// TwinCAT 3 PLC project MotionControl
// ProgramVersion: 3.1.4026.24
// libraries:
//   Tc2_MC2, * (Beckhoff Automation GmbH)
//   Tc2_Standard, * (Beckhoff Automation GmbH)
//   Tc2_SUPS, * (Beckhoff Automation GmbH)
//   Tc2_System, * (Beckhoff Automation GmbH)
//   Tc2_Utilities, * (Beckhoff Automation GmbH)
//   Tc3_DriveMotionControl, * (Beckhoff Automation GmbH)
//   Tc3_IotBase, * (Beckhoff Automation GmbH)
//   Tc3_JsonXml, * (Beckhoff Automation GmbH)
//   Tc3_Module, * (Beckhoff Automation GmbH)
//   VisuDialogs, * (System)
// project tree:
//   / CSVTask.TcTTO, GlobalTextList.TcGTLO, PlcTask.TcTTO, Visualization Manager.TcVMO (not stored)
//   DUTs/ BASIN.TcDUT, BasinStateDisp.TcDUT, HB.TcDUT, MotionType.TcDUT, CTR_SIGNALS_INTERNAL.TcDUT, MOTION_INSTRUCTION.TcDUT, MOTION_FB_STATUS.TcDUT, OUT_SIGNALS.TcDUT, MOTION_CTR.TcDUT, SCRIPTNAME.TcDUT, STATUS.TcDUT
//   GVLs/ GVL_MOTION.TcGVL
//   POUs/ AddCommand.TcPOU, DeleteLastInstruction.TcPOU, ClearScript.TcPOU, DeleteScriptFile.TcPOU, DirectMotion.TcPOU, HomeFixRack.TcPOU, HomeX.TcPOU, HomeY.TcPOU, HomeZ.TcPOU, JsonSaxHandler.TcPOU, MAIN.TcPOU, FunctionBlockMisc.TcPOU, AxisFunctionBlocks.TcPOU, MQTTCOMM.TcPOU, RackCheck.TcPOU, ScriptList.TcPOU, ScriptRead.TcPOU, CSVWrite.TcPOU, ResetAxes.TcPOU, RunCommands.TcPOU, zAxisMoreLogic.TcPOU
//   VISUs/ visMotorControl.TcVIS
// real-time tasks:
//   TASK PlcTask: cycle T#1ms, priority 6, ADS port 350
//   TASK VISU_TASK: cycle T#50000us, priority 14, ADS port 351
//   TASK CSVTask: cycle T#1ms, priority 8, ADS port 353
// motion (NC):
//   TASK NC-Task 1 SAF: cycle T#1ms, priority 4, ADS port 501
//   TASK NC-Task 1 SVB: cycle T#10ms, priority 12, ADS port 511
//   AXIS xAxis (id 1)
//     Dynamic: Acceleration=100, Deceleration=1000, Jerk=4000
//     Velo: RefSearch=10, RefSync=9, FastManual=250, Fast=904.22, Maximum=904.22
//     OtherSettings: AllowMotionCmdToSlave=true, DataPersistence=true
//     encoder EncType=19
//       EncPara: ScaleFactorNumerator=0.0007056311621, MaxCount=#xffffffff
//         Inc: RefSearchInverse=true, RefSyncInverse=false
//     drive DrvType=16
//       DrvPara: MaxCount=#xffffffff, DriveControlDWord=#x00020100
//         Analog: VeloReferenz=994.642, TorqueSetpointScale=10, ScaleFactorActTorque=0.1
//         TimeComp: TaskDelayCycles=1
//     controller CtrType=1
//       CtrPara: PriorControlFactor=1
//         Observer: BandWidth=20
//   AXIS yAxis (id 2)
//     Dynamic: Acceleration=200, Deceleration=2000, Jerk=6000
//     Velo: RefSearch=12, RefSync=5, SlowManual=70, FastManual=300, Fast=452.11, Maximum=452.11
//     OtherSettings: AllowMotionCmdToSlave=true, DataPersistence=true
//     encoder EncType=19
//       EncPara: ScaleFactorNumerator=0.0003125, Inverse=true, MaxCount=#xffffffff
//         Inc: RefSearchInverse=true, RefSyncInverse=false
//     drive DrvType=16
//       DrvPara: Inverse=true, MaxCount=#xffffffff, DriveControlDWord=#x00020100
//         Analog: VeloReferenz=497.321, VeloScale=32, TorqueSetpointScale=10, ScaleFactorActTorque=0.1
//         TimeComp: TaskDelayCycles=1
//     controller CtrType=1
//       CtrPara: PriorControlFactor=1
//         PosDiffControl: Range=10
//         Observer: BandWidth=20
//   AXIS xAxisCoupled (id 3)
//     Dynamic: Acceleration=100, Deceleration=1000, Jerk=4000
//     Velo: RefSearch=10, RefSync=9.0422, SlowManual=45.211, FastManual=271.266, Fast=904.22, Maximum=904.22
//     OtherSettings: AllowMotionCmdToSlave=true, DataPersistence=true
//     encoder EncType=19
//       EncPara: ScaleFactorNumerator=0.0007056311621, Inverse=true, MaxCount=#xffffffff
//         Inc: RefSearchInverse=true, RefSyncInverse=false
//     drive DrvType=16
//       DrvPara: Inverse=true, MaxCount=#xffffffff, DriveControlDWord=#x00020100
//         Analog: VeloReferenz=994.642, TorqueSetpointScale=10, ScaleFactorActTorque=0.1
//         TimeComp: TaskDelayCycles=1
//     controller CtrType=1
//       CtrPara: PriorControlFactor=1
//         PosDiffControl: Range=10
//         Observer: BandWidth=20
//   AXIS zAxis (id 4)
//     Dynamic: Acceleration=200, Deceleration=2000, Jerk=5000
//     Velo: RefSearch=3, RefSync=3, FastManual=200, Fast=22.605, Maximum=210
//     OtherSettings: AllowMotionCmdToSlave=true, DataPersistence=true
//     encoder EncType=19
//       EncPara: ScaleFactorNumerator=0.0003125, Inverse=true, MaxCount=#xffffffff
//         Inc: RefSearchInverse=true, RefSyncInverse=false
//     drive DrvType=16
//       DrvPara: Inverse=true, MaxCount=#xffffffff, DriveControlDWord=#x00020100
//         Analog: VeloReferenz=210, TorqueSetpointScale=10, ScaleFactorActTorque=0.1
//         TimeComp: TaskDelayCycles=1
//     controller CtrType=1
//       CtrPara: PriorControlFactor=1
//         Observer: BandWidth=20
// I/O:
//   DEVICE Device 2 (EtherCAT), AmsNetId 10.1.179.227.3.1
//     Drive 2 (ClearPath EtherCAT Integrated ServoMotor) [ClearPath EC (CoE Rev 2)]
//     Drive 3 (ClearPath EtherCAT Integrated ServoMotor) [ClearPath EC (CoE Rev 2)]
//     Drive 4 (ClearPath EtherCAT Integrated ServoMotor) [ClearPath EC (CoE Rev 2)]
//     Drive 5 (ClearPath EtherCAT Integrated ServoMotor) [ClearPath EC (CoE Rev 2)]
//   DEVICE Device 1 (EtherCAT), AmsNetId 10.1.179.227.2.1
//     Term 1 (EK1200) [EK1200-5000 EtherCAT Power supply (2A E-Bus)]
//       Term 6 (ED2008) [ED2008 | 8-ch. dig. output, 24 V DC, 0.5 A, push-in]
//       Term 7 (ED1008) [ED1008 | 8-ch. dig. input, 24 V DC, 3 ms, push-in]
//       Term 4 (EL9011) [EL9011 End Terminal]
// variable links:
//   NC-Task 1 SAF/Axes/xAxis <-> Device 2 (EtherCAT)/Drive 2 (ClearPath EtherCAT Integrated ServoMotor)
//     Drive/Inputs/In/nDataIn1 <-> TxPDO 2/Following Error Actual Value
//     Drive/Inputs/In/nState1 <-> TxPDO 2/Statusword
//     Drive/Inputs/In/nState2 <-> TxPDO 2/Statusword @bit 8
//     Drive/Inputs/In/nState4 @bit 1 <-> WcState/InputToggle
//     Drive/Inputs/In/nState4 <-> WcState/WcState
//     Drive/Outputs/Out/nCtrl1 <-> RxPDO 2/Controlword
//     Drive/Outputs/Out/nCtrl2 <-> RxPDO 2/Controlword @bit 8
//     Drive/Outputs/Out/nDataOut1 <-> RxPDO 2/Target Position
//     Enc/Inputs/In/nDataIn1 <-> TxPDO 2/Position Actual Value
//     Enc/Inputs/In/nState4 @bit 1 <-> WcState/InputToggle
//     Enc/Inputs/In/nState4 <-> WcState/WcState
//   NC-Task 1 SAF/Axes/xAxisCoupled <-> Device 2 (EtherCAT)/Drive 5 (ClearPath EtherCAT Integrated ServoMotor)
//     Drive/Inputs/In/nDataIn1 <-> TxPDO 2/Following Error Actual Value
//     Drive/Inputs/In/nState1 <-> TxPDO 2/Statusword
//     Drive/Inputs/In/nState2 <-> TxPDO 2/Statusword @bit 8
//     Drive/Inputs/In/nState4 @bit 1 <-> WcState/InputToggle
//     Drive/Inputs/In/nState4 <-> WcState/WcState
//     Drive/Outputs/Out/nCtrl1 <-> RxPDO 2/Controlword
//     Drive/Outputs/Out/nCtrl2 <-> RxPDO 2/Controlword @bit 8
//     Drive/Outputs/Out/nDataOut1 <-> RxPDO 2/Target Position
//     Enc/Inputs/In/nDataIn1 <-> TxPDO 2/Position Actual Value
//     Enc/Inputs/In/nState4 @bit 1 <-> WcState/InputToggle
//     Enc/Inputs/In/nState4 <-> WcState/WcState
//   NC-Task 1 SAF/Axes/yAxis <-> Device 2 (EtherCAT)/Drive 3 (ClearPath EtherCAT Integrated ServoMotor)
//     Drive/Inputs/In/nDataIn1 <-> TxPDO 2/Following Error Actual Value
//     Drive/Inputs/In/nState1 <-> TxPDO 2/Statusword
//     Drive/Inputs/In/nState2 <-> TxPDO 2/Statusword @bit 8
//     Drive/Inputs/In/nState4 @bit 1 <-> WcState/InputToggle
//     Drive/Inputs/In/nState4 <-> WcState/WcState
//     Drive/Outputs/Out/nCtrl1 <-> RxPDO 2/Controlword
//     Drive/Outputs/Out/nCtrl2 <-> RxPDO 2/Controlword @bit 8
//     Drive/Outputs/Out/nDataOut1 <-> RxPDO 2/Target Position
//     Enc/Inputs/In/nDataIn1 <-> TxPDO 2/Position Actual Value
//     Enc/Inputs/In/nState4 @bit 1 <-> WcState/InputToggle
//     Enc/Inputs/In/nState4 <-> WcState/WcState
//   NC-Task 1 SAF/Axes/zAxis <-> Device 2 (EtherCAT)/Drive 4 (ClearPath EtherCAT Integrated ServoMotor)
//     Drive/Inputs/In/nDataIn1 <-> TxPDO 2/Following Error Actual Value
//     Drive/Inputs/In/nState1 <-> TxPDO 2/Statusword
//     Drive/Inputs/In/nState2 <-> TxPDO 2/Statusword @bit 8
//     Drive/Inputs/In/nState4 @bit 1 <-> WcState/InputToggle
//     Drive/Inputs/In/nState4 <-> WcState/WcState
//     Drive/Outputs/Out/nCtrl1 <-> RxPDO 2/Controlword
//     Drive/Outputs/Out/nCtrl2 <-> RxPDO 2/Controlword @bit 8
//     Drive/Outputs/Out/nDataOut1 <-> RxPDO 2/Target Position
//     Enc/Inputs/In/nDataIn1 <-> TxPDO 2/Position Actual Value
//     Enc/Inputs/In/nState4 @bit 1 <-> WcState/InputToggle
//     Enc/Inputs/In/nState4 <-> WcState/WcState
//   MotionControl/MotionControl Instance <-> Device 1 (EtherCAT)/Term 1 (EK1200)/Term 6 (ED2008)
//     PlcTask Outputs/GVL_MOTION.ED2008O/ED2008_Output/MDP5001_200_DO_Channel_{1..8}_Output <-> DO Channel {1..8}/Output  (8 links)
//   MotionControl/MotionControl Instance <-> Device 1 (EtherCAT)/Term 1 (EK1200)/Term 7 (ED1008)
//     PlcTask Inputs/MAIN.ED1008I/ED1008_Input/MDP5001_100_DI_Channel_{1..8}_Input <-> DI Channel {1..8}/Input  (8 links)
//   MotionControl/MotionControl Instance <-> NC-Task 1 SAF/Axes/xAxis
//     PlcTask Inputs/MAIN.xAxis.NcToPlc <-> Outputs/ToPlc
//     PlcTask Outputs/MAIN.xAxis.PlcToNc <-> Inputs/FromPlc
//   MotionControl/MotionControl Instance <-> NC-Task 1 SAF/Axes/xAxisCoupled
//     PlcTask Inputs/MAIN.xAxisCoupled.NcToPlc <-> Outputs/ToPlc
//     PlcTask Outputs/MAIN.xAxisCoupled.PlcToNc <-> Inputs/FromPlc
//   MotionControl/MotionControl Instance <-> NC-Task 1 SAF/Axes/yAxis
//     PlcTask Inputs/MAIN.yAxis.NcToPlc <-> Outputs/ToPlc
//     PlcTask Outputs/MAIN.yAxis.PlcToNc <-> Inputs/FromPlc
//   MotionControl/MotionControl Instance <-> NC-Task 1 SAF/Axes/zAxis
//     PlcTask Inputs/MAIN.zAxis.NcToPlc <-> Outputs/ToPlc
//     PlcTask Outputs/MAIN.zAxis.PlcToNc <-> Inputs/FromPlc

CONFIGURATION MotionControl
    RESOURCE PLC ON TwinCAT3
        TASK CSVTask(INTERVAL := T#1ms, PRIORITY := 8);
        TASK PlcTask(INTERVAL := T#1ms, PRIORITY := 6);
        PROGRAM CSVWrite WITH CSVTask : CSVWrite;
        PROGRAM ScriptRead WITH CSVTask : ScriptRead;
        PROGRAM MAIN WITH PlcTask : MAIN;
    END_RESOURCE
END_CONFIGURATION

// ---- DUTs/BASIN.TcDUT
TYPE BASIN :
STRUCT
	Name	:T_MaxString;
	xMin	:REAL;
	xMax	:REAL;
	yMin	:REAL;
	yMax	:REAL;
END_STRUCT
END_TYPE

// ---- DUTs/BasinStateDisp.TcDUT
{attribute 'qualified_only'}
{attribute 'to_string'}
TYPE BasinStateDisp :
(
	set_xMin	:= 0,
	set_xMax	:= 1,
	set_yMin	:= 2,
	set_yMax	:= 3
);
END_TYPE

// ---- DUTs/HB.TcDUT
TYPE HB :
STRUCT
	HEARTBEAT		:BOOL	:= FALSE; //check in MQTTCOM to keep jog commands online
END_STRUCT
END_TYPE

// ---- DUTs/MotionType.TcDUT
{attribute 'qualified_only'}
{attribute 'to_string'}
TYPE MotionType :
(
	Null			:= 0,
	WaitOK			:= 1,
	Absolute		:= 2,
	Relative		:= 3,
	Time_Wait		:= 4
);
END_TYPE

// ---- DUTs/CTR_SIGNALS_INTERNAL.TcDUT
TYPE CTR_SIGNALS_INTERNAL :
STRUCT
	//motion control signals
	Enable					:BOOL;
	Execute_SPOS			:BOOL;
	Execute_MABS			:BOOL;
	Execute_MREL			:BOOL;
	Execute_RES				:BOOL;
	//Execute_VEL				:BOOL;
	Execute_HALT			:BOOL;
	Execute_STOP			:BOOL;
	Execute_HOME			:BOOL;
	JogFw					:BOOL;
	JogBw					:BOOL;
	JogMode					:E_JogMode;
	SetLocation				:LREAL;
	SetPosition				:LREAL;
	SetVelocity				:LREAL;
	SetAccel				:LREAL;
	LimPos					:BOOL;
	LimNeg					:BOOL;
	IsHoming				:BOOL	:= FALSE;
	
	//axis coupling control
	ExecuteCouple			:BOOL; //connected to GearIn
	ExecuteUncouple			:BOOL; //connected to GearOut
	AxisToCouple			:AXIS_REF;
	
	
END_STRUCT
END_TYPE

// ---- DUTs/MOTION_INSTRUCTION.TcDUT
TYPE MOTION_INSTRUCTION :
STRUCT
	(*motion type*)
	MotionCommand 			:MotionType;
	SetXPosition			:REAL;
	SetXVelocity			:INT := 10;
	SetXAccel				:INT;
	SetYPosition			:REAL;	
	SetYVelocity			:INT := 10;
	SetYAccel				:INT;
	SetZPosition			:REAL;
	SetZVelocity			:INT := 10;
	PauseTime				:TIME;	//comes in as UDINT in MS, variable format T#1D4H5M2S1MS
	Comment					:STRING;
	index					:INT := 0;

END_STRUCT
END_TYPE

// ---- DUTs/MOTION_FB_STATUS.TcDUT
TYPE MOTION_FB_STATUS :
STRUCT
	Status		: BOOL;
	Done		: BOOL;
	Busy		: BOOL;
	Error		: BOOL;
	Active		: BOOL;
	CmdAborted	: BOOL;
	InVelocity	: BOOL;
	ErrorID		: UDINT;

END_STRUCT
END_TYPE

// ---- DUTs/OUT_SIGNALS.TcDUT
TYPE OUT_SIGNALS :
STRUCT
	PowerError				:BOOL;
	MoveActive				:BOOL;
	MoveDone				:BOOL;
	VelocityOut				:LREAL;
	PositionOut				:LREAL;
	HaltDone				:BOOL;
	AxisCoupled				:BOOL;
	SetPosDone				:BOOL;
END_STRUCT
END_TYPE

// ---- DUTs/MOTION_CTR.TcDUT
TYPE MOTION_CTR :
STRUCT
	CMDHOME					:BOOL	:= FALSE; //run home routine
	CMDHOMEX				:BOOL	:= FALSE;
	CMDHOMEY				:BOOL	:= FALSE;
	CMDHOMEZ				:BOOL	:= FALSE;
	SETXPOS					:BOOL	:= FALSE;
	MOVEX					:BOOL	:= FALSE;
	POSX					:LREAL	:= 0;
	SETYPOS					:BOOL	:= FALSE;
	MOVEY					:BOOL	:= FALSE;
	POSY					:LREAL	:= 0;
	SETZPOS					:BOOL	:= FALSE;
	MOVEZ					:BOOL	:= FALSE;
	POSZ					:LREAL	:= 0;
	
	//CMDSETZLIM			:BOOL	:= FALSE; //this will set the safe lower limit of z to where it is currently positioned
	//CMDFINDSTOPS			:BOOL	:= FALSE; //run find stops routine
	CMDCOUPLE				:BOOL	:= FALSE; //cycle between couple and uncouple x axes
	STOP					:BOOL	:= FALSE; //pause motion during script run if true. set to false to continue motion
	AXESEN					:BOOL	:= FALSE; //sends enable signal to all axes
	AXESRESET				:BOOL	:= FALSE; //reset each axis, reset home and hardstop states
	BRAKEREL				:BOOL	:= FALSE;
	
	CMDADD					:BOOL	:= FALSE; //add instruction to script
	CMDCLR					:BOOL	:= FALSE; //clear script
	CMDSCRIPTDEL			:BOOL	:= FALSE; //delete script file
	CMDDEL					:BOOL	:= FALSE; //delete instruction at end of script
	CMDLOOP					:BOOL	:= FALSE; //sets script to run indefinitely and forces separate data files for each script run
	CMDRUN					:BOOL	:= FALSE; //run script if all safety conditions are met (homed, hard stops located, x axes coupled, safe z set)
	CMDCSVRESET				:BOOL	:= FALSE; //reset csvwrite logic CHANGED
	CMDSCRIPTWRITE			:BOOL	:= FALSE; //write script to file based on script name entered
	CMDSCRIPTREAD			:BOOL	:= FALSE; //read script from file based on script name
	CMDREQLIST				:BOOL	:= FALSE;
	CMDREQSCRIPT			:BOOL	:= FALSE;
	SCRIPTITERATIONS		:INT	:= 1; //number of times a script will be executed in a run
	SCRIPTNAME				:T_MaxString; //name of script for data and script files.
	BASINCTR				:BOOL	:= FALSE; //true = basin A, false = basin B CHANGED

	XJOGFW					:BOOL	:= FALSE;
	XJOGBW					:BOOL	:= FALSE;
	YJOGFW					:BOOL	:= FALSE;
	YJOGBW					:BOOL	:= FALSE;
	ZJOGFW					:BOOL	:= FALSE;
	ZJOGBW					:BOOL	:= FALSE;
END_STRUCT
END_TYPE

// ---- DUTs/SCRIPTNAME.TcDUT
TYPE SCRIPTNAME :
STRUCT
	payload		:T_MaxString;	
	start		:BOOL	:= FALSE;
	end			:BOOL	:= FALSE;		
END_STRUCT
END_TYPE

// ---- DUTs/STATUS.TcDUT
TYPE STATUS :
STRUCT
	MoveActive			:BOOL;
	eStop				:BOOL;
	
	Rack_Err			:BOOL	:= FALSE;
	Script_Open_Err		:BOOL	:= FALSE;	
	Script_Read_Err		:BOOL	:= FALSE;
	List_Overflow_Err	:BOOL	:= FALSE;
	Move_Rel_Err		:BOOL 	:= FALSE;
	Move_Abs_Err		:BOOL	:= FALSE;
	//HS_Err				:BOOL	:= FALSE;
	Basin_Exceed_Err	:BOOL	:= FALSE;
	//Basin_Set_Err		:BOOL	:= FALSE;
	
	
	AxesLocated			:BOOL	:= FALSE;
	//HardStopLoc			:BOOL	:= FALSE; 
	//zSafeSet			:BOOL	:= FALSE;
	//BasinSet			:BOOL	:= FALSE;
	Stop_Int			:BOOL	:= FALSE; //for display only
	PowerError			:BOOL	:= FALSE;
	
	CurInstr			:INT;
	NextInstr			:INT;
	ScriptEnd			:INT;
	RUN_INDEX			:INT;
	
	xCoupled			:BOOL;
	xPosOut				:LREAL;
	xVelOut				:LREAL;
	yPosOut				:LREAL;
	yVelOut				:LREAL;
	zPosOut				:LREAL;
	zVelOut				:LREAL;
	
	basinxMin			:LREAL;
	basinxMax			:LREAL;
	basinyMin			:LREAL;
	basinyMax			:LREAL;
	basinstate			:INT	:= 0;

	
	HardStopLocations	:ARRAY[0..2] OF LREAL	:= [100000,8991,1000]; //includes carriage offsets 
	CARRIAGE_OFFSETS	:ARRAY[0..2] OF LREAL	:= [500,250,100]; //for display. also in GVL_MOTION
	
	
END_STRUCT
END_TYPE

// ---- GVLs/GVL_MOTION.TcGVL
//variables must be referenced GVL_MOTION.etc b/c of attribute
//persistent data causes problems when changing variable declarations
{attribute 'qualified_only'}
VAR_GLOBAL
	//motor control signals
	
	xCon					:CTR_SIGNALS_INTERNAL;
	xcCon					:CTR_SIGNALS_INTERNAL;
	yCon					:CTR_SIGNALS_INTERNAL;
	zCon					:CTR_SIGNALS_INTERNAL;
	
	xJogFW					:BOOL;
	xJogBW					:BOOL;
	yJogFW					:BOOL;
	yJogBW					:BOOL;
	zJogFW					:BOOL;
	zJogBW					:BOOL;
	
	MOVEXYZ					:BOOL;
	
	ED2008O AT %Q*			:ED2008_46D0FC69;
	Z_BRAKE_OFF				:BOOL;
	
	//external controls
	STOP_EXT				:BOOL;
	STOP_INT				:BOOL; //control signal
	EXT_CTR					:MOTION_CTR; 
	TEST_CTR				:MOTION_CTR; //test buffer for MQTT
	HB						:HB;
	{attribute 'TcEncoding':='UTF-8'}
	TopicRcv				:STRING(255); //for MQTT
	
	//script variables
	
	InstructionBuffer		:MOTION_INSTRUCTION; //set externally (MQTT) or locally
	TestBuffer				:MOTION_INSTRUCTION; //test buffer for MQTT
	EmptyInstruction		:MOTION_INSTRUCTION;
	Script 					:ARRAY[0..99] OF MOTION_INSTRUCTION; //add commands from instruction buffer or load script
	ScriptReadBuffer		:ARRAY[0..99] OF MOTION_INSTRUCTION; //buffer for ScriptRead
	ContinuousMode			:BOOL; //override number of script runs and run until set false
	ScriptEnd				:INT						:= 0; //empty/not executed
	InstructionState		:INT						:= 0; //control case statement in RunCommands
	TxtBxWaitOK				:BOOL						:= TRUE; //hide text box
	HaltMem					:BOOL						:= FALSE; //part of the waitOK motion button control
	
	
	STATUS					:STATUS;
	ActiveBasin				:BASIN;
	BasinA					:BASIN	:= (Name := 'BasinA',
										xMin := 0,			
										xMax := 100000,
										yMin := 0,
										yMax := 5000);
	
	BasinB					:BASIN	:= (Name := 'BasinB',
										xMin := 0,			
										xMax := 100000,
										yMin := 5050,
										yMax := 8991);
	BASINLAMPA				:BOOL;
	BASINLAMPB				:BOOL;
	CSV_ROW					:INT						:= 0;
	
	//variables for script list
	
	LISTSTART				:BOOL						:= FALSE;
	LISTEND					:BOOL						:= FALSE;
	LIST					:ARRAY[0..999] OF T_MaxString;
	LISTCNT					:INT						:= 0;
	SCRIPTNAME				:SCRIPTNAME;
	
	//filelistp				:VISU_FBFileListProvider;
	
	xOut					:OUT_SIGNALS;
	xCOut					:OUT_SIGNALS;
	yOut					:OUT_SIGNALS;	
	zOut					:OUT_SIGNALS;
	xHomeStatus				:MOTION_FB_STATUS;
	xCHomeStatus			:MOTION_FB_STATUS;
	yHomeStatus				:MOTION_FB_STATUS;
	zHomeStatus				:MOTION_FB_STATUS;
	
	CurInstruction			:INT						:= 0; //current instruction
	NextInstruction			:INT; //only for display
	RUN_INDEX				:INT						:= 1; //increment after script run
	
	//for the drop down lists
	
	xyzCMDSelect			:ARRAY[0..4] OF MotionType	:= [0,1,2,3,4];
	
	//safety controls

	zSafeSet				:BOOL						:= FALSE;
	zSafeDisable			:BOOL						:= FALSE; 	(*in zAxisMoreLogic*)
	zSafePosition			:LREAL						:= 0;	
	
	//homing variables
	
	HomingState				:INT						:= 0;
	RevCouplePrep			:BOOL						:= FALSE;
	//x and y stage from rail to top of y stage
	//z stage from rail to bottom of z stage
	CARRIAGE_OFFSETS		:ARRAY[0..2] OF LREAL		:= [500,250,100]; //also in STATUS
END_VAR

VAR_GLOBAL
	AxesLocated				:BOOL						:= FALSE;
	xLocated				:BOOL						:= FALSE;
	yLocated				:BOOL						:= FALSE;
	zLocated				:BOOL						:= FALSE;
							
END_VAR

// ---- POUs/CSVWrite.TcPOU
(* Writing of CSV file in text mode. None of the field value is containing any non-printing control characters like line feed, carriage return, quotation marks, semicolon... *)
PROGRAM CSVWrite
VAR
	index			:INT; //write script for loop
	step			:DWORD 			:= 0;(*state control*)
	//datawrite		:BOOL			:= FALSE;(*start by writing header, then set TRUE*)
	scriptwrite		:BOOL			:= FALSE;(*write column headers then script*)
	headerstep		:INT			:= 0;(*state control for header write*)
	datastep		:INT			:= 0;(*state control for data write*)
	
	bWrite			:BOOL			:= FALSE;(* Rising edge starts program execution *)
	sNetId			:T_AmsNetId		:= '';	(* TwinCAT system network address *)
	bBusy			:BOOL;
	bError			:BOOL;
	nErrId			:UDINT;
	
	nRow	 		:UDINT 			:= 0;(* Row number (record) *)
	nPassCompare	:UDINT			:= 0;
	nColumn			:UDINT 			:= 0;(* Column number (record field) *)
	hFile			:UINT			:= 0;(* File handle of the source file *)
	
	fbFileOpen		:FB_FileOpen;(* Opens file *)
	fbFileClose		:FB_FileClose;(* Closes file *)
	fbFilePuts		:FB_FilePuts;(* Writes one record (line) *)
	fbWriter		:FB_CSVMemBufferWriter;(* Helper function block used to create CSV data bytes (single record line) *)
	fbCMD			:NT_StartProcess; //run CMD to create data directories
	
	sCSVLine		:T_MaxString	:= '';(* Single CSV text line (row, record), we are using string as record buffer (your are able to see created fields) *)
	sCSVField		:T_MaxString	:= '';(* Single CSV field value (column, record field) *)

	TEMP			:T_MaxString	:= '';
	CMDPATH			:T_MaxString	:= 'C:\Windows\System32\cmd.exe';
	COMNDLINE		:T_MaxString	:= '/C "mkdir '; // /C carries out command string then terminates
	TOPDIR			:T_MaxString	:= 'C:\';
	FILENAME		:T_MaxString;
	FILEPATH		:T_MaxString; 	//path of directory for current experiment including file name	
	HOLDNAME_M		:T_MaxString;	//save file name for appending data - Massa
	HOLDNAME_K		:T_MaxString;	//save file name for appending data - Keyence
	HOLDNAME_S		:T_MaxString;	//save file name for appending data - Sonar
	
	fbTime			:FB_LocalSystemTime;
	timestring		:STRING;
END_VAR

//TODO 2 modes: write data and write script
fbtime(bEnable := TRUE, dwCycle := 1);

//write data controls are internal, read and write script controls are external
DEFAULT_CSV_FIELD_SEP := 16#2C;(* Comma ASCII code *)
//DEFAULT_CSV_FIELD_SEP := 16#3B;(* Semicolon ASCII code *)

IF GVL_MOTION.EXT_CTR.CMDCSVRESET THEN
	GVL_MOTION.EXT_CTR.CMDCSVRESET			:= FALSE;
	bWrite								:= FALSE;
	step								:= 0;
	headerstep							:= 0;
	datastep							:= 0;
	//datawrite							:= FALSE;
	scriptwrite							:= FALSE;
	index								:= 0;
	GVL_MOTION.CSV_ROW					:= 0;
	//GVL_DAQ.CSV_PASS_COMPARE			:= 0;
END_IF



IF GVL_MOTION.EXT_CTR.CMDSCRIPTWRITE THEN
	GVL_MOTION.EXT_CTR.CMDSCRIPTWRITE	:= FALSE;
	scriptwrite							:= FALSE;
	//GVL_DAQ.DAQ_CTR_INT.CSVWriteMode	:= CSVWriteMode.script;
	bWrite								:= TRUE;
END_IF

CASE step OF
	0:	(* Wait for rising edge at bWrite variable *)
		IF bWrite THEN
			//GVL_DAQ.DAQ_CTR_INT.CSVWriteMode	:= CSVWriteMode.keyence; //TEST ONLY
			bBusy 					:= TRUE;
			bError					:= FALSE;
			nErrId					:= 0;
			hFile					:= 0;
			nRow					:= 0;
			nColumn					:= 0;
			TOPDIR					:= 'C:\';
			//make sure C:\MOTION_SCRIPTS exists
			fbCMD( PATHSTR:= CMDPATH, DIRNAME:= 'C:\', COMNDLINE:= concat(COMNDLINE, 'MOTION_SCRIPTS"'), START:= TRUE);
			fbCMD(START:= FALSE);
			IF NOT fbCMD.BUSY THEN
				bWrite 					:= FALSE;
				FILEPATH				:= '';
				step 					:= 1;
			END_IF
		END_IF
		
	1:
	
		TOPDIR						:= concat(TOPDIR, 'MOTION_SCRIPTS\');
		FILENAME					:= concat(GVL_MOTION.EXT_CTR.SCRIPTNAME, '_Script.csv');
		
		//path to working folder
		FILEPATH	:= concat(TOPDIR, FILENAME);	
		step:=2;
		
		
	2:	(* Open source file *)
		fbFileOpen(  bExecute := FALSE  );
		//header to be written - open at beginning
		
		fbFileOpen( sNetId := sNetId, sPathName := FILEPATH, nMode := FOPEN_MODEWRITE OR FOPEN_MODETEXT,
					ePath := PATH_GENERIC, bExecute := TRUE );
				
		step := 3;
	
	3:(* Wait until open not busy *)
		fbFileOpen( bExecute := FALSE, bError => bError, nErrID => nErrID, hFile => hFile );
		IF NOT fbFileOpen.bBusy THEN
			IF NOT fbFileOpen.bError THEN
				step := 4;
				//TODO add to step 4 for write script
			ELSE(* Error: file not found? *)
				step := 100;
				
			END_IF
		END_IF

	4:(* write header (if not datawrite), then write data *)
		sCSVLine := '';
		fbWriter.eCmd := eEnumCmd_First;(* Write first field value *)
		
		
		 //script write
			IF NOT scriptwrite THEN //header
				CASE headerstep OF
				0:
					sCSVField				:= STRING_TO_CSVFIELD('Basin', FALSE);	
					fbWriter( 	pBuffer := ADR( sCSVLine ), cbBuffer := SIZEOF( sCSVLine ) - 1, putValue := sCSVField, pValue := 0, cbValue := 0,
									bCRLF := FALSE );(* bCRLF == TRUE => Write CRLF after the last field value *)
					IF fbWriter.bOk THEN
						fbWriter.eCmd 		:= eEnumCmd_Next;(* Write next field value *)
					ELSE(* Error *)
						step := 100;
						RETURN;
					END_IF		
					sCSVField	:= STRING_TO_CSVFIELD('x Min', FALSE);	
					fbWriter( 	pBuffer := ADR( sCSVLine ), cbBuffer := SIZEOF( sCSVLine ) - 1, putValue := sCSVField, pValue := 0, cbValue := 0,
									bCRLF := FALSE );(* bCRLF == TRUE => Write CRLF after the last field value *)
					sCSVField	:= STRING_TO_CSVFIELD('x Max', FALSE);	
					fbWriter( 	pBuffer := ADR( sCSVLine ), cbBuffer := SIZEOF( sCSVLine ) - 1, putValue := sCSVField, pValue := 0, cbValue := 0,
									bCRLF := FALSE );(* bCRLF == TRUE => Write CRLF after the last field value *)	
					sCSVField	:= STRING_TO_CSVFIELD('y Min', FALSE);	
					fbWriter( 	pBuffer := ADR( sCSVLine ), cbBuffer := SIZEOF( sCSVLine ) - 1, putValue := sCSVField, pValue := 0, cbValue := 0,
									bCRLF := FALSE );(* bCRLF == TRUE => Write CRLF after the last field value *)
					sCSVField	:= STRING_TO_CSVFIELD('y Max', FALSE);	
					fbWriter( 	pBuffer := ADR( sCSVLine ), cbBuffer := SIZEOF( sCSVLine ) - 1, putValue := sCSVField, pValue := 0, cbValue := 0,
									bCRLF := TRUE );(* bCRLF == TRUE => Write CRLF after the last field value *)	
					headerstep			:= 1;
				1:
					sCSVField				:= STRING_TO_CSVFIELD(GVL_MOTION.ActiveBasin.Name, FALSE);	
					fbWriter( 	pBuffer := ADR( sCSVLine ), cbBuffer := SIZEOF( sCSVLine ) - 1, putValue := sCSVField, pValue := 0, cbValue := 0,
									bCRLF := FALSE );(* bCRLF == TRUE => Write CRLF after the last field value *)
					IF fbWriter.bOk THEN
						fbWriter.eCmd 		:= eEnumCmd_Next;(* Write next field value *)
					ELSE(* Error *)
						step := 100;
						RETURN;
					END_IF		
					sCSVField	:= STRING_TO_CSVFIELD(REAL_TO_STRING(GVL_MOTION.ActiveBasin.xMin), FALSE);	
					fbWriter( 	pBuffer := ADR( sCSVLine ), cbBuffer := SIZEOF( sCSVLine ) - 1, putValue := sCSVField, pValue := 0, cbValue := 0,
									bCRLF := FALSE );(* bCRLF == TRUE => Write CRLF after the last field value *)
					sCSVField	:= STRING_TO_CSVFIELD(REAL_TO_STRING(GVL_MOTION.ActiveBasin.xMax), FALSE);	
					fbWriter( 	pBuffer := ADR( sCSVLine ), cbBuffer := SIZEOF( sCSVLine ) - 1, putValue := sCSVField, pValue := 0, cbValue := 0,
									bCRLF := FALSE );(* bCRLF == TRUE => Write CRLF after the last field value *)	
					sCSVField	:= STRING_TO_CSVFIELD(REAL_TO_STRING(GVL_MOTION.ActiveBasin.yMin), FALSE);	
					fbWriter( 	pBuffer := ADR( sCSVLine ), cbBuffer := SIZEOF( sCSVLine ) - 1, putValue := sCSVField, pValue := 0, cbValue := 0,
									bCRLF := FALSE );(* bCRLF == TRUE => Write CRLF after the last field value *)
					sCSVField	:= STRING_TO_CSVFIELD(REAL_TO_STRING(GVL_MOTION.ActiveBasin.yMax), FALSE);	
					fbWriter( 	pBuffer := ADR( sCSVLine ), cbBuffer := SIZEOF( sCSVLine ) - 1, putValue := sCSVField, pValue := 0, cbValue := 0,
									bCRLF := TRUE );(* bCRLF == TRUE => Write CRLF after the last field value *)	
					headerstep			:= 2;	
				2:
					sCSVField				:= STRING_TO_CSVFIELD('Command', FALSE);	
					fbWriter( 	pBuffer := ADR( sCSVLine ), cbBuffer := SIZEOF( sCSVLine ) - 1, putValue := sCSVField, pValue := 0, cbValue := 0,
									bCRLF := FALSE );(* bCRLF == TRUE => Write CRLF after the last field value *)
					IF fbWriter.bOk THEN
						fbWriter.eCmd 		:= eEnumCmd_Next;(* Write next field value *)
					ELSE(* Error *)
						step := 100;
						RETURN;
					END_IF			
					sCSVField	:= STRING_TO_CSVFIELD('x Pos', FALSE);
					fbWriter( 	pBuffer := ADR( sCSVLine ), cbBuffer := SIZEOF( sCSVLine ) - 1, putValue := sCSVField, pValue := 0, cbValue := 0,
									bCRLF := FALSE );(* bCRLF == TRUE => Write CRLF after the last field value *)	
					sCSVField	:= STRING_TO_CSVFIELD('x Vel', FALSE);
					fbWriter( 	pBuffer := ADR( sCSVLine ), cbBuffer := SIZEOF( sCSVLine ) - 1, putValue := sCSVField, pValue := 0, cbValue := 0,
									bCRLF := FALSE );(* bCRLF == TRUE => Write CRLF after the last field value *)	
					sCSVField	:= STRING_TO_CSVFIELD('y Pos', FALSE);
					fbWriter( 	pBuffer := ADR( sCSVLine ), cbBuffer := SIZEOF( sCSVLine ) - 1, putValue := sCSVField, pValue := 0, cbValue := 0,
									bCRLF := FALSE );(* bCRLF == TRUE => Write CRLF after the last field value *)	
					sCSVField	:= STRING_TO_CSVFIELD('y Vel', FALSE);
					fbWriter( 	pBuffer := ADR( sCSVLine ), cbBuffer := SIZEOF( sCSVLine ) - 1, putValue := sCSVField, pValue := 0, cbValue := 0,
									bCRLF := FALSE );(* bCRLF == TRUE => Write CRLF after the last field value *)	
					sCSVField	:= STRING_TO_CSVFIELD('z Pos', FALSE);
					fbWriter( 	pBuffer := ADR( sCSVLine ), cbBuffer := SIZEOF( sCSVLine ) - 1, putValue := sCSVField, pValue := 0, cbValue := 0,
									bCRLF := FALSE );(* bCRLF == TRUE => Write CRLF after the last field value *)	
					sCSVField	:= STRING_TO_CSVFIELD('z Vel', FALSE);
					fbWriter( 	pBuffer := ADR( sCSVLine ), cbBuffer := SIZEOF( sCSVLine ) - 1, putValue := sCSVField, pValue := 0, cbValue := 0,
									bCRLF := FALSE );(* bCRLF == TRUE => Write CRLF after the last field value *)
					sCSVField	:= STRING_TO_CSVFIELD('Pause Time', FALSE);
					fbWriter( 	pBuffer := ADR( sCSVLine ), cbBuffer := SIZEOF( sCSVLine ) - 1, putValue := sCSVField, pValue := 0, cbValue := 0,
									bCRLF := FALSE );(* bCRLF == TRUE => Write CRLF after the last field value *)	
					sCSVField	:= STRING_TO_CSVFIELD('Comment', FALSE);
					fbWriter( 	pBuffer := ADR( sCSVLine ), cbBuffer := SIZEOF( sCSVLine ) - 1, putValue := sCSVField, pValue := 0, cbValue := 0,
									bCRLF := TRUE );(* bCRLF == TRUE => Write CRLF after the last field value *)
					
					headerstep			:= 0;
					scriptwrite			:= TRUE;
				END_CASE
				IF RIGHT( sCSVLine, 2 ) = '$R$L' THEN
						sCSVLine := REPLACE( sCSVLine, '$L', 2, LEN( sCSVLine ) - 1 );
				END_IF
				step					:= 5;	
			ELSE //write script
				IF index <= 99 THEN
					IF GVL_MOTION.Script[index].MotionCommand = MotionType.Null THEN
						index			:= 0;
						step			:= 10;
					ELSE
						sCSVField	:= STRING_TO_CSVFIELD(TO_STRING(GVL_MOTION.Script[index].MotionCommand), FALSE);
						fbWriter( 	pBuffer := ADR( sCSVLine ), cbBuffer := SIZEOF( sCSVLine ) - 1, putValue := sCSVField, pValue := 0, cbValue := 0,
									bCRLF := FALSE );(* bCRLF == TRUE => Write CRLF after the last field value *)
						IF fbWriter.bOk THEN
							fbWriter.eCmd := eEnumCmd_Next;(* Write next field value *)
						ELSE(* Error *)
							step 		:= 100;
							RETURN;
						END_IF
							
						sCSVField	:= STRING_TO_CSVFIELD(REAL_TO_STRING(GVL_MOTION.Script[index].SetXPosition), FALSE);
						fbWriter( 	pBuffer := ADR( sCSVLine ), cbBuffer := SIZEOF( sCSVLine ) - 1, putValue := sCSVField, pValue := 0, cbValue := 0,
									bCRLF := FALSE );(* bCRLF == TRUE => Write CRLF after the last field value *)
						sCSVField	:= STRING_TO_CSVFIELD(INT_TO_STRING(GVL_MOTION.Script[index].SetXVelocity), FALSE);
						fbWriter( 	pBuffer := ADR( sCSVLine ), cbBuffer := SIZEOF( sCSVLine ) - 1, putValue := sCSVField, pValue := 0, cbValue := 0,
									bCRLF := FALSE );(* bCRLF == TRUE => Write CRLF after the last field value *)	
						sCSVField	:= STRING_TO_CSVFIELD(REAL_TO_STRING(GVL_MOTION.Script[index].SetYPosition), FALSE);
						fbWriter( 	pBuffer := ADR( sCSVLine ), cbBuffer := SIZEOF( sCSVLine ) - 1, putValue := sCSVField, pValue := 0, cbValue := 0,
									bCRLF := FALSE );(* bCRLF == TRUE => Write CRLF after the last field value *)
						sCSVField	:= STRING_TO_CSVFIELD(INT_TO_STRING(GVL_MOTION.Script[index].SetYVelocity), FALSE);
						fbWriter( 	pBuffer := ADR( sCSVLine ), cbBuffer := SIZEOF( sCSVLine ) - 1, putValue := sCSVField, pValue := 0, cbValue := 0,
									bCRLF := FALSE );(* bCRLF == TRUE => Write CRLF after the last field value *)	
						sCSVField	:= STRING_TO_CSVFIELD(REAL_TO_STRING(GVL_MOTION.Script[index].SetZPosition), FALSE);
						fbWriter( 	pBuffer := ADR( sCSVLine ), cbBuffer := SIZEOF( sCSVLine ) - 1, putValue := sCSVField, pValue := 0, cbValue := 0,
									bCRLF := FALSE );(* bCRLF == TRUE => Write CRLF after the last field value *)
						sCSVField	:= STRING_TO_CSVFIELD(INT_TO_STRING(GVL_MOTION.Script[index].SetZVelocity), FALSE);
						fbWriter( 	pBuffer := ADR( sCSVLine ), cbBuffer := SIZEOF( sCSVLine ) - 1, putValue := sCSVField, pValue := 0, cbValue := 0,
									bCRLF := FALSE );(* bCRLF == TRUE => Write CRLF after the last field value *)	
						sCSVField	:= STRING_TO_CSVFIELD(TIME_TO_STRING(GVL_MOTION.Script[index].PauseTime), FALSE);
						fbWriter( 	pBuffer := ADR( sCSVLine ), cbBuffer := SIZEOF( sCSVLine ) - 1, putValue := sCSVField, pValue := 0, cbValue := 0,
									bCRLF := FALSE );(* bCRLF == TRUE => Write CRLF after the last field value *)
						sCSVField	:= STRING_TO_CSVFIELD(GVL_MOTION.Script[index].Comment, FALSE);
						fbWriter( 	pBuffer := ADR( sCSVLine ), cbBuffer := SIZEOF( sCSVLine ) - 1, putValue := sCSVField, pValue := 0, cbValue := 0,
									bCRLF := TRUE );(* bCRLF == TRUE => Write CRLF after the last field value *)
						IF RIGHT( sCSVLine, 2 ) = '$R$L' THEN
							sCSVLine		:= REPLACE( sCSVLine, '$L', 2, LEN( sCSVLine ) - 1 );
						END_IF
						index				:= index + 1;
						step				:= 5;			
					END_IF
					
				ELSE
						index				:= 0;
						step				:= 10;
				END_IF
				
			END_IF
			
		

	5:(* Write single text line *)
		fbFilePuts( bExecute := FALSE );
		fbFilePuts( sNetId := sNetId, hFile := hFile, sLine := sCSVLine, bExecute := TRUE );
		step := 6;

	6:(* Wait until write not busy *)
		fbFilePuts( bExecute := FALSE, bError => bError, nErrID => nErrID );
		IF NOT fbFilePuts.bBusy THEN
			IF NOT fbFilePuts.bError THEN
				step := 4;(* Write next record *)
			ELSE(* Error *)
				step := 100;
			END_IF
		END_IF

	10:	(* Close source file *)
		fbFileClose( bExecute := FALSE );
		fbFileClose( sNetId := sNetId, hFile := hFile, bExecute := TRUE );
		step := 11;

	11:(* Wait until close not busy *)
		fbFileClose( bExecute := FALSE, bError => bError, nErrID => nErrID );
		IF ( NOT fbFileClose.bBusy ) THEN
			hFile := 0;
			step := 100;
		END_IF

	100: (* Error or ready step => cleanup *)
		IF ( hFile <> 0 ) THEN
			step := 10; (* Close the source file *)
		ELSE
			bBusy := FALSE;
		
			step := 0;	(* Ready *)
		END_IF

END_CASE

END_PROGRAM

// ---- POUs/ScriptRead.TcPOU
(* Reading of CSV file in text mode. None of the field value is containing any non-printing control characters like line feed, carriage return, quotation marks, semicolon... *)
PROGRAM ScriptRead
VAR
	sNetId			:T_AmsNetId := '';	(* TwinCAT system network address *)
	FilePath		:T_MaxString := 'C:\data\';(* CSV source file path and name *)
	sCSVLine		:T_MaxString := '';(* Single CSV text line (row, record), we are using string as record buffer (your are able to see read fields)  *)
	sCSVField		:T_MaxString := '';(* Single CSV field value (column, record field) *)
	
	bRead			:BOOL	:= FALSE;(* Rising edge starts program execution *)
	bBusy			:BOOL;
	bError			:BOOL;
	nErrId			:UDINT;
	nRow	 		:UDINT 	:= 0;(* Row number (record) *)
	nColumn			:UDINT 	:= 0;(* Column number (record field) *)
	hFile			:UINT	:= 0;(* File handle of the source file *)
	step			:DWORD 	:= 0;
	fbFileOpen		:FB_FileOpen;(* Opens file *)
	fbFileClose		:FB_FileClose;(* Closes file *)
	fbFileGets		:FB_FileGets;(* Reads one record (line) *)
	fbReader		:FB_CSVMemBufferReader;(* Helper function block used to parse CSV data bytes (single record line) *)
	lastline		:UDINT;
	temp			:ARRAY[0..100, 0..12 ] OF STRING;
END_VAR

IF GVL_MOTION.EXT_CTR.CMDSCRIPTREAD THEN
	GVL_MOTION.EXT_CTR.CMDSCRIPTREAD				:= FALSE;
	bRead											:= TRUE;
END_IF

CASE step OF
	0:	(* Wait for rising edge at bRead variable *)
		IF bRead THEN
			bRead 		:= FALSE;
			bBusy 		:= TRUE;
			bError		:= FALSE;
			GVL_MOTION.STATUS.Script_Open_Err	:= FALSE; //pop up in HMI
			GVL_MOTION.STATUS.Script_Read_Err	:= FALSE; //pop up in HMI
			nErrId		:= 0;
			hFile		:= 0;
			FilePath	:= 'C:\data\';
			FilePath	:= concat(FilePath, GVL_MOTION.Basin.Name);
			FilePath	:= concat(FilePath, '\');
			FilePath	:= concat(FilePath, GVL_MOTION.EXT_CTR.SCRIPTNAME);
			FilePath	:= concat(FilePath, '_');
			FilePath	:= concat(FilePath, 'Script.csv');
			lastline	:= 100;
			nRow		:= 0;
			nColumn		:= 0;
			MEMSET( ADR( GVL_MOTION.ScriptReadBuffer ), 0, SIZEOF( GVL_MOTION.ScriptReadBuffer ) );
			MEMSET( ADR( temp ), 0, SIZEOF( temp ) );
			step 		:= 1;
		END_IF
	

	1:	(* Open source file *)
		fbFileOpen(  bExecute := FALSE  );
		fbFileOpen( sNetId := sNetId, sPathName := FilePath, nMode := FOPEN_MODEREAD OR FOPEN_MODETEXT,(* Open file in TEXT mode! *)
					ePath := PATH_GENERIC, bExecute := TRUE );
		step := 2;

	2:(* Wait until open not busy *)
		fbFileOpen( bExecute := FALSE, bError => bError, nErrID => nErrID, hFile => hFile );
		IF NOT fbFileOpen.bBusy THEN
			IF NOT fbFileOpen.bError THEN
				step := 3;
			ELSE(* Error: file not found? *)
				GVL_MOTION.STATUS.Script_Open_Err	:= TRUE;
				step := 100;
				
			END_IF
		END_IF

	3:	(* Read single line (record) *)
		fbFileGets( bExecute := FALSE );
		fbFileGets( sNetId := sNetId, hFile := hFile, bExecute := TRUE );
		step := 4;

	4:(* Wait until read not busy *)
		fbFileGets( bExecute := FALSE, bError => bError, nErrID => nErrID, sLine => sCSVLine );
		IF NOT fbFileGets.bBusy THEN
			IF NOT fbFileGets.bError THEN
				IF fbFileGets.bEOF THEN
					lastline	:= nRow - 1;
					nRow		:= 3; //skip labels on script verify
					step := 6;(* End of file reached => check and load script *)
				ELSE

					(* FB_FileGets returns text line without the CR (carriage return) character.
					We have to restore the CR character (replace the $L character with $R$L characters) *)
					IF RIGHT( sCSVLine, 1 ) = '$L' THEN
						sCSVLine := REPLACE( sCSVLine, '$R$L', 2, LEN( sCSVLine ) );
					END_IF

					step := 5;
				END_IF
			ELSE(* Error *)
				step := 100;
			END_IF
		END_IF

	5:(* Parse single line (record) *)
		fbReader.eCmd := eEnumCmd_First;(* Read first field value *)
		REPEAT
			fbReader( pBuffer := ADR( sCSVLine ), cbBuffer := SIZEOF( sCSVLine ), getValue => sCSVField );
			IF fbReader.bOk THEN
				fbReader.eCmd := eEnumCmd_Next;(* Read next field value *)

				IF ( nRow <= 102 ) THEN
					IF ( nColumn <= 12 ) THEN
						temp[nRow, nColumn] := CSVFIELD_TO_STRING( sCSVField, FALSE );(* TODO: Save or use the field value in your application *)
					END_IF
				END_IF

				nColumn := nColumn + 1;(* Increment number of read columns *)
				IF fbReader.bCRLF THEN(* CRLF == TRUE => End of reacord reached *)
					nRow 		:= nRow + 1;(* Increment number of read records *)
					nColumn 	:= 0;(* Reset number of columns *)
				END_IF

			ELSE(* Error: End of record reached or all fields read *)
				step := 3;(* Try to read next line *)
			END_IF
		UNTIL NOT fbReader.bOk
		END_REPEAT
		
	6:
		GVL_MOTION.Basin.Name	:= temp[1,0];
		GVL_MOTION.Basin.xMin	:= STRING_TO_LREAL(temp[1,1]);
		GVL_MOTION.Basin.xMax	:= STRING_TO_LREAL(temp[1,2]);
		GVL_MOTION.Basin.yMin	:= STRING_TO_LREAL(temp[1,3]);
		GVL_MOTION.Basin.yMax	:= STRING_TO_LREAL(temp[1,4]);
		step	:= 7;
			
	
	7: (*check format and write script*)
 		IF nRow <= lastline THEN
			IF temp[nRow, 0] = 'Absolute' THEN
				GVL_MOTION.ScriptReadBuffer[nRow - 3].MotionCommand	:= MotionType.Absolute;
			ELSIF temp[nRow, 0] = 'Relative' THEN
				GVL_MOTION.ScriptReadBuffer[nRow - 3].MotionCommand	:= MotionType.Relative;
			ELSIF temp[nRow, 0] = 'WaitOk' THEN
				GVL_MOTION.ScriptReadBuffer[nRow - 3].MotionCommand	:= MotionType.WaitOK;
			ELSE
				GVL_MOTION.STATUS.Script_Read_Err	:= TRUE;
				step							:= 10;
			END_IF	
			
			IF temp[nRow, 1] = 'Manual' THEN
				GVL_MOTION.ScriptReadBuffer[nRow - 3].zType	:= zBehavior.Manual;
			ELSIF temp[nRow, 1] = 'SedSurface' THEN
				GVL_MOTION.ScriptReadBuffer[nRow - 3].MotionCommand	:= zBehavior.SedSurface;
			ELSIF temp[nRow, 1] = 'WaterSurface' THEN
				GVL_MOTION.ScriptReadBuffer[nRow - 3].MotionCommand	:= zBehavior.WaterSurface;
			ELSE
				GVL_MOTION.STATUS.Script_Read_Err	:= TRUE;
				step							:= 10;
			END_IF	
			
			IF temp[nRow, 2] = 'none' THEN
				GVL_MOTION.ScriptReadBuffer[nRow - 3].DataTrigger	:= DataTrigger.none;
			ELSIF temp[nRow, 2] = 'timed' THEN
				GVL_MOTION.ScriptReadBuffer[nRow - 3].DataTrigger	:= DataTrigger.timed;
			ELSIF temp[nRow, 2] = 'x' THEN
				GVL_MOTION.ScriptReadBuffer[nRow - 3].DataTrigger	:= DataTrigger.x;
			ELSIF temp[nRow, 2] = 'y' THEN
				GVL_MOTION.ScriptReadBuffer[nRow - 3].DataTrigger	:= DataTrigger.y;
			ELSIF temp[nRow, 2] = 'z' THEN
				GVL_MOTION.ScriptReadBuffer[nRow - 3].DataTrigger	:= DataTrigger.z;
			ELSE
				GVL_MOTION.STATUS.Script_Read_Err	:= TRUE;
				step							:= 10;
			END_IF	
			
			IF temp[nRow, 3] = '' THEN
				;
			ELSIF temp[nRow, 3] = 'KSM' THEN
				GVL_MOTION.ScriptReadBuffer[nRow - 3].Acq_Keyence	:= TRUE;
				GVL_MOTION.ScriptReadBuffer[nRow - 3].Acq_Sonar		:= TRUE;
				GVL_MOTION.ScriptReadBuffer[nRow - 3].Acq_Massa		:= TRUE;
			ELSIF temp[nRow, 3] = 'KS' THEN
				GVL_MOTION.ScriptReadBuffer[nRow - 3].Acq_Keyence	:= TRUE;
				GVL_MOTION.ScriptReadBuffer[nRow - 3].Acq_Sonar		:= TRUE;
			ELSIF temp[nRow, 3] = 'KM' THEN
				GVL_MOTION.ScriptReadBuffer[nRow - 3].Acq_Keyence	:= TRUE;
				GVL_MOTION.ScriptReadBuffer[nRow - 3].Acq_Massa		:= TRUE;
			ELSIF temp[nRow, 3] = 'SM' THEN
				GVL_MOTION.ScriptReadBuffer[nRow - 3].Acq_Sonar		:= TRUE;
				GVL_MOTION.ScriptReadBuffer[nRow - 3].Acq_Massa		:= TRUE;
			ELSIF temp[nRow, 3] = 'K' THEN
				GVL_MOTION.ScriptReadBuffer[nRow - 3].Acq_Keyence	:= TRUE;
			ELSIF temp[nRow, 3] = 'S' THEN
				GVL_MOTION.ScriptReadBuffer[nRow - 3].Acq_Sonar		:= TRUE;
			ELSIF temp[nRow, 3] = 'M' THEN
				GVL_MOTION.ScriptReadBuffer[nRow - 3].Acq_Massa		:= TRUE;	
			ELSE
				GVL_MOTION.STATUS.Script_Read_Err	:= TRUE;
				step							:= 10;
			END_IF	
			
			IF ( (0 <= STRING_TO_INT(temp[nRow, 4]) ) AND
   			(STRING_TO_INT(temp[nRow, 4]) <= GVL_MOTION.STATUS.HardStopLocations[0]) ) THEN
				GVL_MOTION.ScriptReadBuffer[nRow - 3].SetXPosition	:= STRING_TO_REAL(temp[nRow, 4]);			
			ELSE
				GVL_MOTION.STATUS.Script_Read_Err	:= TRUE;
				step							:= 10;
			END_IF	 
			
			IF ( (0 <= STRING_TO_INT(temp[nRow, 5]) ) AND
   			(STRING_TO_INT(temp[nRow, 5]) <= 300) ) THEN
				GVL_MOTION.ScriptReadBuffer[nRow - 3].SetXVelocity	:= STRING_TO_INT(temp[nRow, 5]);			
			ELSE
				GVL_MOTION.STATUS.Script_Read_Err	:= TRUE;
				step							:= 10;
			END_IF
			
			IF ( (0 <= STRING_TO_INT(temp[nRow, 6]) ) AND
   			(STRING_TO_INT(temp[nRow, 6]) <= GVL_MOTION.STATUS.HardStopLocations[1]) ) THEN
				GVL_MOTION.ScriptReadBuffer[nRow - 3].SetYPosition	:= STRING_TO_REAL(temp[nRow, 6]);			
			ELSE
				GVL_MOTION.STATUS.Script_Read_Err	:= TRUE;
				step							:= 10;
			END_IF	 
			
			IF ( (0 <= STRING_TO_INT(temp[nRow, 7]) ) AND
   			(STRING_TO_INT(temp[nRow, 7]) <= 300) ) THEN
				GVL_MOTION.ScriptReadBuffer[nRow - 3].SetYVelocity	:= STRING_TO_INT(temp[nRow, 7]);			
			ELSE
				GVL_MOTION.STATUS.Script_Read_Err	:= TRUE;
				step							:= 10;
			END_IF
			
			IF ( (0 <= STRING_TO_INT(temp[nRow, 8]) ) AND
   			(STRING_TO_INT(temp[nRow, 8]) <= GVL_MOTION.STATUS.HardStopLocations[2]) ) THEN
				GVL_MOTION.ScriptReadBuffer[nRow - 3].SetZPosition	:= STRING_TO_REAL(temp[nRow, 8]);			
			ELSE
				GVL_MOTION.STATUS.Script_Read_Err	:= TRUE;
				step							:= 10;
			END_IF	 
			
			IF ( (0 <= STRING_TO_INT(temp[nRow, 9]) ) AND
   			(STRING_TO_INT(temp[nRow, 9]) <= 30) ) THEN
				GVL_MOTION.ScriptReadBuffer[nRow - 3].SetZVelocity	:= STRING_TO_INT(temp[nRow, 9]);			
			ELSE
				GVL_MOTION.STATUS.Script_Read_Err	:= TRUE;
				step							:= 10;
			END_IF
			
			GVL_MOTION.ScriptReadBuffer[nRow - 3].PauseTime			:= STRING_TO_TIME(temp[nRow, 10]);
			
			GVL_MOTION.ScriptReadBuffer[nRow - 3].Comment				:= temp[nRow, 11];
			
			nRow	:= nRow + 1;
		ELSE //no errors found
			ClearScript();
			GVL_MOTION.ScriptEnd				:= UDINT_TO_INT(nRow - 1);
			GVL_MOTION.Script					:= GVL_MOTION.ScriptReadBuffer;
			
			step	:= 10;	
		END_IF

	10:	(* Close source file *)
		fbFileClose( bExecute := FALSE );
		fbFileClose( sNetId := sNetId, hFile := hFile, bExecute := TRUE );
		step := 11;

	11:(* Wait until close not busy *)
		fbFileClose( bExecute := FALSE, bError => bError, nErrID => nErrID );
		IF ( NOT fbFileClose.bBusy ) THEN
			hFile := 0;
			step := 100;
		END_IF

	100: (* Error or ready step => cleanup *)
		IF ( hFile <> 0 ) THEN
			step := 10; (* Close the source file *)
		ELSE
			bBusy := FALSE;
			step := 0;	(* Ready *)
		END_IF

END_CASE

END_PROGRAM

// ---- POUs/ClearScript.TcPOU
PROGRAM ClearScript
VAR
END_VAR

IF GVL_MOTION.EXT_CTR.CMDCLR THEN
	GVL_MOTION.EXT_CTR.CMDCLR	:= FALSE;
	GVL_MOTION.EXT_CTR.CMDRUN 	:= FALSE;
	GVL_MOTION.ScriptEnd 		:= 0;
	GVL_MOTION.CurInstruction 	:= 0;
	GVL_MOTION.InstructionState := 0;
	GVL_MOTION.HaltMem 			:= FALSE;
	GVL_MOTION.TxtBxWaitOK 		:= TRUE;
	MEMSET(ADR(GVL_MOTION.Script), 0, SIZEOF(GVL_MOTION.Script));
END_IF

END_PROGRAM

// ---- POUs/MAIN.TcPOU
PROGRAM MAIN
VAR
	xAxis					:AXIS_REF;
	xAxisCoupled			:AXIS_REF;
	yAxis					:AXIS_REF;
	zAxis					:AXIS_REF;
		
	xAxisFunctions			:AxisFunctionBlocks;
	xCoupledFunctions		:AxisFunctionBlocks;
	yAxisFunctions			:AxisFunctionBlocks;
	zAxisFunctions			:AxisFunctionBlocks;
	
	ED1008I AT %I*			:ED1008_AB7978D6; //current or voltage input
	
	DM						:BOOL;
	couplestate				:INT	:= 0;
	basintoggle				:BOOL;
	boot_done				:BOOL	:= FALSE;
	
	xNearStop				:BOOL	:= FALSE;
	yNearStop				:BOOL	:= FALSE;

END_VAR

//external/mqtt control signals located in gvl's as struct EXT_CTR
//100 instruction script. modify in GVL_MOTION and RunCommands()

//digital io and internal variable assignments
GVL_MOTION.xCon.LimNeg				 		:= NOT(ED1008I.ED1008_Input.MDP5001_100_DI_Channel_1_Input);
GVL_MOTION.yCon.LimPos				 		:= NOT(ED1008I.ED1008_Input.MDP5001_100_DI_Channel_2_Input);
GVL_MOTION.xCon.LimPos				 		:= NOT(ED1008I.ED1008_Input.MDP5001_100_DI_Channel_3_Input);
GVL_MOTION.zCon.LimPos				 		:= NOT(ED1008I.ED1008_Input.MDP5001_100_DI_Channel_4_Input);
GVL_MOTION.xcCon.LimNeg				 		:= NOT(ED1008I.ED1008_Input.MDP5001_100_DI_Channel_5_Input);
GVL_MOTION.zCon.LimNeg				 		:= NOT(ED1008I.ED1008_Input.MDP5001_100_DI_Channel_6_Input);
GVL_MOTION.yCon.LimNeg				 		:= NOT(ED1008I.ED1008_Input.MDP5001_100_DI_Channel_7_Input);
GVL_MOTION.STOP_EXT							:= NOT(ED1008I.ED1008_Input.MDP5001_100_DI_Channel_8_Input);

GVL_MOTION.ED2008O.ED2008_Output.MDP5001_200_DO_Channel_7_Output	:= GVL_MOTION.Z_BRAKE_OFF;

GVL_MOTION.NextInstruction					:= GVL_MOTION.CurInstruction + 1;

//alternative position read
//xPos 										:= xAxis.NcToPlc.ActPos;

//external variable assignments
GVL_MOTION.xCon.JogFw						:= GVL_MOTION.EXT_CTR.XJOGFW OR GVL_MOTION.xJogFW;
GVL_MOTION.xCon.JogBw						:= GVL_MOTION.EXT_CTR.XJOGBW OR GVL_MOTION.xJogBW;
GVL_MOTION.yCon.JogFw						:= GVL_MOTION.EXT_CTR.YJOGFW OR GVL_MOTION.yJogFW;
GVL_MOTION.yCon.JogBw						:= GVL_MOTION.EXT_CTR.YJOGBW OR GVL_MOTION.yJogBW;
GVL_MOTION.zCon.JogFw						:= GVL_MOTION.EXT_CTR.ZJOGFW OR GVL_MOTION.zJogFW;
GVL_MOTION.zCon.JogBw						:= GVL_MOTION.EXT_CTR.ZJOGBW OR GVL_MOTION.zJogBW;

GVL_MOTION.STATUS.CurInstr					:= GVL_MOTION.CurInstruction;
GVL_MOTION.STATUS.NextInstr					:= GVL_MOTION.NextInstruction;
GVL_MOTION.STATUS.ScriptEnd					:= GVL_MOTION.ScriptEnd;
GVL_MOTION.STATUS.RUN_INDEX					:= GVL_MOTION.RUN_INDEX;
GVL_MOTION.STATUS.xCoupled					:= GVL_MOTION.xOut.AxisCoupled;

GVL_MOTION.STATUS.xVelOut					:= GVL_MOTION.xOut.VelocityOut;
GVL_MOTION.STATUS.yVelOut					:= GVL_MOTION.yOut.VelocityOut;

GVL_MOTION.STATUS.zPosOut					:= GVL_MOTION.zOut.PositionOut + GVL_MOTION.CARRIAGE_OFFSETS[2];
GVL_MOTION.STATUS.zVelOut					:= GVL_MOTION.zOut.VelocityOut;
GVL_MOTION.STATUS.AxesLocated				:= GVL_MOTION.AxesLocated;
//GVL_MOTION.STATUS.zSafeSet					:= GVL_MOTION.zSafeSet;			
//GVL_MOTION.STATUS.HaltDone					:= GVL_MOTION.xOut.HaltDone;
GVL_MOTION.STATUS.PowerError				:= GVL_MOTION.xOut.PowerError OR GVL_MOTION.yOut.PowerError	OR
											   GVL_MOTION.zOut.PowerError OR GVL_MOTION.xCOut.PowerError;	

CASE GVL_MOTION.STATUS.basinstate OF
0:
	GVL_MOTION.ActiveBasin					:= GVL_MOTION.BasinA;
	GVL_MOTION.BASINLAMPA					:= TRUE;
	GVL_MOTION.BASINLAMPB					:= FALSE;
	IF GVL_MOTION.EXT_CTR.BASINCTR THEN
		GVL_MOTION.EXT_CTR.BASINCTR			:= FALSE;
		GVL_MOTION.STATUS.basinstate		:= 1;
	END_IF
1:
	GVL_MOTION.ActiveBasin					:= GVL_MOTION.BasinB;
	GVL_MOTION.BASINLAMPA					:= FALSE;
	GVL_MOTION.BASINLAMPB					:= TRUE;
	IF GVL_MOTION.EXT_CTR.BASINCTR THEN
		GVL_MOTION.EXT_CTR.BASINCTR			:= FALSE;
		GVL_MOTION.STATUS.basinstate		:= 0;
	END_IF	

END_CASE
											   
GVL_MOTION.STATUS.basinxMin					:= GVL_MOTION.ActiveBasin.xMin;
GVL_MOTION.STATUS.basinxMax					:= GVL_MOTION.ActiveBasin.xMax;
GVL_MOTION.STATUS.basinyMin					:= GVL_MOTION.ActiveBasin.yMin;
GVL_MOTION.STATUS.basinyMax					:= GVL_MOTION.ActiveBasin.yMax;
										   						   
IF  GVL_MOTION.xOut.PositionOut + GVL_MOTION.CARRIAGE_OFFSETS[0] >= GVL_MOTION.ActiveBasin.xMin 
AND GVL_MOTION.xOut.PositionOut + GVL_MOTION.CARRIAGE_OFFSETS[0] <= GVL_MOTION.ActiveBasin.xMax 
THEN
	GVL_MOTION.STATUS.xPosOut				:= GVL_MOTION.xOut.PositionOut + GVL_MOTION.CARRIAGE_OFFSETS[0];
	IF NOT (GVL_MOTION.xCon.Execute_HOME OR GVL_MOTION.EXT_CTR.CMDHOME OR xNearStop) THEN
			GVL_MOTION.xCon.JogMode			:= MC_JOGMODE_STANDARD_FAST;
		ELSE
			GVL_MOTION.xCon.JogMode			:= MC_JOGMODE_STANDARD_SLOW;
	END_IF
ELSE
	GVL_MOTION.STATUS.xPosOut				:= -999999;
	GVL_MOTION.xCon.JogMode					:= MC_JOGMODE_STANDARD_SLOW;
END_IF

IF  GVL_MOTION.yOut.PositionOut + GVL_MOTION.CARRIAGE_OFFSETS[1] >= GVL_MOTION.ActiveBasin.yMin 
AND GVL_MOTION.yOut.PositionOut + GVL_MOTION.CARRIAGE_OFFSETS[1] <= GVL_MOTION.ActiveBasin.yMax 
THEN
	IF basintoggle THEN
		GVL_MOTION.yJogBW					:= FALSE;
		GVL_MOTION.yJogFW					:= FALSE;
		GVL_MOTION.EXT_CTR.YJOGBW			:= FALSE;
		GVL_MOTION.EXT_CTR.YJOGFW			:= FALSE;
		basintoggle							:= FALSE;
	END_IF
	GVL_MOTION.STATUS.yPosOut				:= GVL_MOTION.yOut.PositionOut + GVL_MOTION.CARRIAGE_OFFSETS[1];
	IF NOT (GVL_MOTION.yCon.Execute_HOME OR GVL_MOTION.EXT_CTR.CMDHOME OR yNearStop) THEN
			GVL_MOTION.yCon.JogMode			:= MC_JOGMODE_STANDARD_FAST;
		ELSE
			GVL_MOTION.yCon.JogMode			:= MC_JOGMODE_STANDARD_SLOW;
	END_IF
ELSE
	IF NOT basintoggle THEN
		GVL_MOTION.yJogBW					:= FALSE;
		GVL_MOTION.yJogFW					:= FALSE;
		GVL_MOTION.EXT_CTR.YJOGBW			:= FALSE;
		GVL_MOTION.EXT_CTR.YJOGFW			:= FALSE;
		basintoggle							:= TRUE;		
	END_IF
	GVL_MOTION.STATUS.yPosOut				:= -999999;
	GVL_MOTION.yCon.JogMode					:= MC_JOGMODE_STANDARD_SLOW;
END_IF	
	
//increasing jog speed may cause axis to lock up if it crashes into end stop
//pulse jog off at changeover to force reclick and new speed
//jogmode for x and y set above in basin coordinates control
IF GVL_MOTION.STATUS.HardStopLocations[0] - GVL_MOTION.STATUS.xPosOut < 600
OR GVL_MOTION.STATUS.xPosOut - GVL_MOTION.CARRIAGE_OFFSETS[0] < 600
THEN
	xNearStop								:= TRUE;
	IF GVL_MOTION.xCon.JogMode = MC_JOGMODE_STANDARD_FAST THEN
		GVL_MOTION.xJogBW					:= FALSE;
		GVL_MOTION.xJogFW					:= FALSE;
		GVL_MOTION.EXT_CTR.XJOGBW			:= FALSE;
		GVL_MOTION.EXT_CTR.XJOGFW			:= FALSE;
	END_IF
ELSE
	xNearStop								:= FALSE;
	IF GVL_MOTION.xCon.JogMode = MC_JOGMODE_STANDARD_SLOW THEN
		GVL_MOTION.xJogBW					:= FALSE;
		GVL_MOTION.xJogFW					:= FALSE;
		GVL_MOTION.EXT_CTR.XJOGBW			:= FALSE;
		GVL_MOTION.EXT_CTR.XJOGFW			:= FALSE;
	END_IF
END_IF

IF GVL_MOTION.STATUS.HardStopLocations[1] - GVL_MOTION.STATUS.yPosOut < 300
OR GVL_MOTION.STATUS.yPosOut - GVL_MOTION.CARRIAGE_OFFSETS[1] < 300 
THEN
	yNearStop								:= TRUE;
	IF GVL_MOTION.yCon.JogMode = MC_JOGMODE_STANDARD_FAST THEN
		GVL_MOTION.yJogBW					:= FALSE;
		GVL_MOTION.yJogFW					:= FALSE;
		GVL_MOTION.EXT_CTR.YJOGBW			:= FALSE;
		GVL_MOTION.EXT_CTR.YJOGFW			:= FALSE;
	END_IF
ELSE
	yNearStop								:= FALSE;
	IF GVL_MOTION.yCon.JogMode = MC_JOGMODE_STANDARD_SLOW THEN
		GVL_MOTION.yJogBW					:= FALSE;
		GVL_MOTION.yJogFW					:= FALSE;
		GVL_MOTION.EXT_CTR.YJOGBW			:= FALSE;
		GVL_MOTION.EXT_CTR.YJOGFW			:= FALSE;
	END_IF	
END_IF

// IF GVL_MOTION.STATUS.HardStopLocations[2] - GVL_MOTION.STATUS.zPosOut < 150
// OR GVL_MOTION.STATUS.zPosOut - GVL_MOTION.CARRIAGE_OFFSETS[2] < 150 
// THEN
// 	IF GVL_MOTION.zCon.JogMode = MC_JOGMODE_STANDARD_FAST THEN
// 		GVL_MOTION.zJogBW					:= FALSE;
// 		GVL_MOTION.zJogFW					:= FALSE;
// 	END_IF
// 	GVL_MOTION.zCon.JogMode					:= MC_JOGMODE_STANDARD_SLOW;
// ELSE
// 	IF GVL_MOTION.zCon.JogMode = MC_JOGMODE_STANDARD_SLOW THEN
// 		GVL_MOTION.zJogBW					:= FALSE;
// 		GVL_MOTION.zJogFW					:= FALSE;
// 	END_IF
// 	GVL_MOTION.zCon.JogMode					:= MC_JOGMODE_STANDARD_FAST;
// END_IF
GVL_MOTION.zCon.JogMode					:= MC_JOGMODE_STANDARD_FAST;			

//coupled axis assignments, modify as needed for additional coupled axes
//xAxis
GVL_MOTION.xCon.AxisToCouple 				:= xAxisCoupled;
IF GVL_MOTION.EXT_CTR.CMDCOUPLE THEN
	GVL_MOTION.EXT_CTR.CMDCOUPLE			:= FALSE;
	CASE couplestate OF
		0: 
		GVL_MOTION.xCon.ExecuteUncouple		:= FALSE;
		GVL_MOTION.xCon.ExecuteCouple		:= TRUE;
		couplestate							:= 1;
		1:
		GVL_MOTION.xCon.ExecuteCouple		:= FALSE;
		GVL_MOTION.xCon.ExecuteUncouple		:= TRUE;
		couplestate							:= 0;
	END_CASE

END_IF		   						   

//axis function blocks
xAxisFunctions(Axis:=xAxis,
			   Control:=GVL_MOTION.xCon,
			   Output:=GVL_MOTION.xOut,
			   HomeStatus:=GVL_MOTION.xHomeStatus);	
xCoupledFunctions(Axis:=xAxisCoupled,
				  Control:=GVL_MOTION.xcCon,
				  Output:=GVL_MOTION.xCOut,
				  HomeStatus:=GVL_MOTION.xCHomeStatus);
yAxisFunctions(Axis:=yAxis,
			   Control:=GVL_MOTION.yCon,
			   Output:=GVL_MOTION.yOut,
			   HomeStatus:=GVL_MOTION.yHomeStatus);
zAxisFunctions(Axis:=zAxis,
			   Control:=GVL_MOTION.zCon,
			   Output:=GVL_MOTION.zOut,
			   HomeStatus:=GVL_MOTION.zHomeStatus);	
			   
//additional logic for axisfunctionblocks
FunctionBlockMisc(); 

//mqtt communication functions for external control/gui
MQTTCOMM();

//reset all axes from error state and reset several function state variables
ResetAxes();

//axis control signals currently tied to VISU
zAxisMoreLogic();

//generate list of script titles
ScriptList();

//delete script based on selected name
DeleteScriptFile();

HomeX(); //TODO need xccon limneg logic

HomeY();

HomeZ();

IF GVL_MOTION.EXT_CTR.SETXPOS THEN
	GVL_MOTION.EXT_CTR.SETXPOS				:= FALSE;
	GVL_MOTION.xCon.SetLocation				:= GVL_MOTION.EXT_CTR.POSX - GVL_MOTION.CARRIAGE_OFFSETS[0];
	GVL_MOTION.xCon.Execute_SPOS			:= TRUE;
END_IF
IF GVL_MOTION.xOut.SetPosDone THEN
	GVL_MOTION.xLocated						:= TRUE;
	GVL_MOTION.xCon.Execute_SPOS			:= FALSE;	
END_IF

IF GVL_MOTION.EXT_CTR.SETYPOS THEN
	GVL_MOTION.EXT_CTR.SETYPOS				:= FALSE;
	GVL_MOTION.yCon.SetLocation				:= GVL_MOTION.EXT_CTR.POSY - GVL_MOTION.CARRIAGE_OFFSETS[1];
	GVL_MOTION.yCon.Execute_SPOS			:= TRUE;
END_IF
IF GVL_MOTION.yOut.SetPosDone THEN
	GVL_MOTION.yLocated						:= TRUE;
	GVL_MOTION.yCon.Execute_SPOS			:= FALSE;	
END_IF

IF GVL_MOTION.EXT_CTR.SETZPOS THEN
	GVL_MOTION.EXT_CTR.SETZPOS				:= FALSE;
	GVL_MOTION.zCon.SetLocation				:= GVL_MOTION.EXT_CTR.POSZ - GVL_MOTION.CARRIAGE_OFFSETS[2];
	GVL_MOTION.zCon.Execute_SPOS			:= TRUE;
END_IF
IF GVL_MOTION.zOut.SetPosDone THEN
	GVL_MOTION.zLocated						:= TRUE;
	GVL_MOTION.zCon.Execute_SPOS			:= FALSE;	
END_IF

IF GVL_MOTION.xLocated AND GVL_MOTION.yLocated AND GVL_MOTION.zLocated THEN
	GVL_MOTION.AxesLocated					:= TRUE;
END_IF

//needs to come after set position or axis reset is executed
//HardStopsNew();

//script control logic						 
AddCommand();
ClearScript();
DeleteLastInstruction();

//require safe z limit, home complete, x axes coupled, hard stops located, basin set
//check before RunCommands is executed
// IF (NOT GVL_MOTION.AxesLocated)
// OR (NOT GVL_MOTION.xOut.AxisCoupled) //OR (NOT GVL_MOTION.STATUS.HardStopLoc) 
// THEN
// 	GVL_MOTION.CurInstruction				:= 0;
// 	GVL_MOTION.EXT_CTR.CMDRUN				:= FALSE;	//maybe change this to internal variable
// END_IF

IF NOT GVL_MOTION.EXT_CTR.CMDRUN AND GVL_MOTION.AxesLocated AND GVL_MOTION.xOut.AxisCoupled THEN
	DM										:= TRUE;
	DirectMotion();
ELSE
	DM										:= FALSE;	
END_IF

IF GVL_MOTION.EXT_CTR.CMDRUN AND GVL_MOTION.AxesLocated AND GVL_MOTION.xOut.AxisCoupled
AND NOT DM THEN
	RunCommands(); //toggler
ELSE
	GVL_MOTION.CurInstruction				:= 0;
	GVL_MOTION.InstructionState				:= 0;
END_IF

IF GVL_MOTION.EXT_CTR.STOP THEN
	GVL_MOTION.EXT_CTR.STOP					:= FALSE;
END_IF

END_PROGRAM

// ---- POUs/AxisFunctionBlocks.TcPOU
FUNCTION_BLOCK AxisFunctionBlocks
VAR_IN_OUT
	Axis					:AXIS_REF;	
	Control					:CTR_SIGNALS_INTERNAL;
	Output					:OUT_SIGNALS;
	HomeStatus				:MOTION_FB_STATUS;
END_VAR	
VAR
	//function blocks
	mcPower					:MC_Power;
	mcSetPosition			:MC_SetPosition;
	mcMoveAbsolute			:MC_MoveAbsolute;
	mcMoveRelative			:MC_MoveRelative;
	mcMoveVelocity			:MC_MoveVelocity;
	mcReset					:MC_Reset;
	mcHalt					:MC_Halt;
	mcStop					:MC_Stop;
	mcReadActualVelocity	:MC_ReadActualVelocity;
	mcReadActualPosition	:MC_ReadActualPosition;
	mcJog					:MC_Jog;
	mcHome					:MC_Home;	
	mcGearIn				:MC_GearIn;
	mcGearOut				:MC_GearOut;
END_VAR
VAR // added by the converter: edge detectors and wires of the graphical bodies
    _w1, _w5, _w6, _w8, _w11 : BOOL;
    _w2, _w3, _w4, _w7, _w9, _w10 : ANY;
END_VAR

mcPower(Axis := Axis, Enable := _w1, Enable_Positive := NOT Control.LimPos AND _w1, Enable_Negative := _w2); // MC_Power
Output.MoveActive := _w3;
mcMoveAbsolute(
    Axis := Axis,
    Execute := _w4,
    Position := Control.SetPosition,
    Velocity := Control.SetVelocity); // MC_MoveAbsolute
Output.SetPosDone := mcSetPosition.Done;
_w7 := _w5 AND _w6;
mcReset(Axis := Axis, Execute := Control.Execute_RES); // MC_Reset
_w1 := _w8 AND GVL_MOTION.AXESEN_INT;
mcMoveRelative(
    Axis := Axis,
    Execute := _w9,
    Distance := Control.SetPosition,
    Velocity := Control.SetVelocity); // MC_MoveRelative
_w4 := mcPower.Status AND Control.Execute_MABS;
_w8 := NOT GVL_MOTION.STATUS.eStop;
Output.MoveDone := _w10;
_w3 := mcMoveAbsolute.Active OR mcMoveRelative.Active;
_w9 := mcPower.Status AND Control.Execute_MREL;
mcStop(Axis := Axis, Execute := Control.Execute_STOP); // MC_Stop
mcHome(Axis := Axis, Execute := Control.Execute_HOME, bCalibrationCam := Control.LimNeg); // MC_Home
_w5 := NOT Control.IsHoming;
_w2 := _w7 OR _w11;
Output.HaltDone := mcHalt.Done;
_w6 := NOT Control.LimNeg;
_w11 := Control.IsHoming AND _w1;
Output.PowerError := mcPower.Error;
mcGearIn(Master := Axis, Slave := Control.AxisToCouple, Execute := Control.ExecuteCouple); // MC_GearIn
mcSetPosition(Axis := Axis, Execute := Control.Execute_SPOS, Position := Control.SetLocation); // MC_SetPosition
mcReadActualVelocity(Axis := Axis, Enable := GVL_MOTION.AXESEN_INT); // MC_ReadActualVelocity
Output.VelocityOut := mcReadActualVelocity.ActualVelocity;
HomeStatus.Busy := mcHome.Busy;
HomeStatus.Active := mcHome.Active;
HomeStatus.CmdAborted := mcHome.CommandAborted;
HomeStatus.Error := mcHome.Error;
HomeStatus.ErrorID := mcHome.ErrorID;
mcReadActualPosition(Axis := Axis, Enable := GVL_MOTION.AXESEN_INT); // MC_ReadActualPosition
HomeStatus.Done := mcHome.Done;
mcHalt(Axis := Axis, Execute := Control.Execute_HALT); // MC_Halt
mcJog(Axis := Axis, JogForward := Control.JogFw, JogBackwards := Control.JogBw, Mode := Control.JogMode); // MC_Jog
_w10 := mcMoveRelative.Done OR mcMoveAbsolute.Done;
Output.PositionOut := mcReadActualPosition.Position;
Output.AxisCoupled := mcGearIn.InGear;
mcGearOut(Slave := Control.AxisToCouple, Execute := Control.ExecuteUncouple); // MC_GearOut

END_FUNCTION_BLOCK

// ---- POUs/FunctionBlockMisc.TcPOU
PROGRAM FunctionBlockMisc
VAR

	FB_WritePersistentData_0: FB_WritePersistentData;
	TON_0: TON;
	TON_1: TON;
	NotBusy: BOOL;
	//1 second ups function writes data and performs quick shutdown
	//check on input SPDM_VAR_BOOST - saves different task data on different PLC cycles?
	FB_S_UPS_BAPI_0: FB_S_UPS_BAPI; 
END_VAR

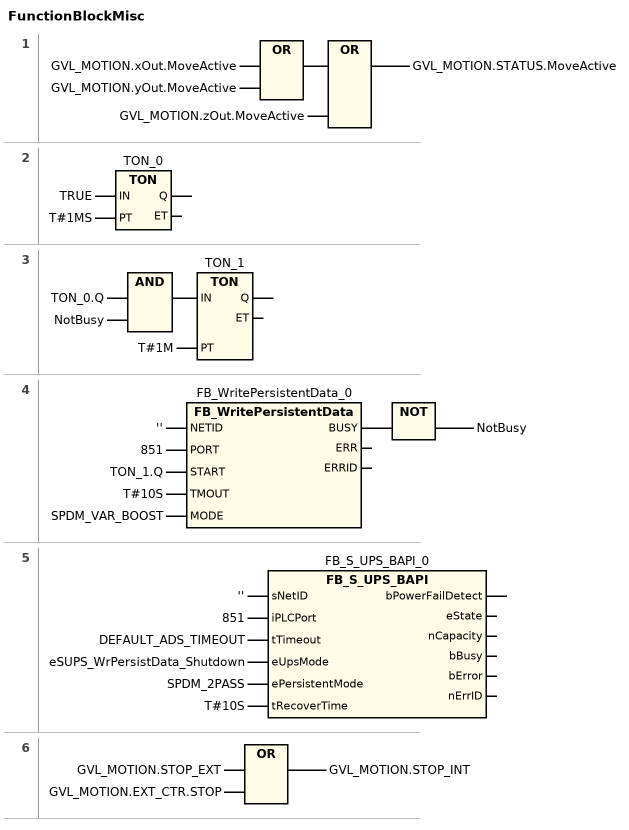
// NETWORK 1
GVL_MOTION.STATUS.MoveActive := (GVL_MOTION.xOut.MoveActive OR GVL_MOTION.yOut.MoveActive) OR GVL_MOTION.zOut.MoveActive;

// NETWORK 2
TON_0(IN := TRUE, PT := T#1MS); // TON

// NETWORK 3
TON_1(IN := TON_0.Q AND NotBusy, PT := T#1M); // TON

// NETWORK 4
FB_WritePersistentData_0(NETID := '', PORT := 851, START := TON_1.Q, TMOUT := T#10S, MODE := SPDM_VAR_BOOST); // FB_WritePersistentData
NotBusy := NOT FB_WritePersistentData_0.BUSY;

// NETWORK 5
FB_S_UPS_BAPI_0(
    sNetID := '',
    iPLCPort := 851,
    tTimeout := DEFAULT_ADS_TIMEOUT,
    eUpsMode := eSUPS_WrPersistData_Shutdown,
    ePersistentMode := SPDM_2PASS,
    tRecoverTime := T#10S); // FB_S_UPS_BAPI

// NETWORK 6
GVL_MOTION.STOP_INT := GVL_MOTION.STOP_EXT OR GVL_MOTION.EXT_CTR.STOP;

END_PROGRAM

// ---- POUs/MQTTCOMM.TcPOU
PROGRAM MQTTCOMM
VAR
    fbMqttClient    :FB_IotMqttClient;
    bSetParameter   :BOOL 		 	:= TRUE;
    bConnect        :BOOL 		 	:= TRUE;	
	
	(* published message *)
	
	MotionStatusPub :STRING(255)	:= 'MOTION/STATUS';
	MotionCTREcho	:STRING(255)	:= 'MOTION/CTR_ECHO';
	MotionINSTREcho	:STRING(255)	:= 'MOTION/INSTR_ECHO';
	HBEcho			:STRING(255)	:= 'MOTION/HB_ECHO';

	ScriptSend		:STRING(255)	:= 'MOTION/SCRIPTSEND';
	ScriptNames		:STRING(255)	:= 'MOTION/SCRIPTNAMES';
	sPayloadPub 	:STRING(1000);
	fbTimer 		:TON			:= (PT:=T#500MS);
	HBtimer 		:TON			:= (PT:=T#1S);
	scriptTimer		:TON			:= (PT:=T#2MS);
	found 			:UDINT;	
	notreset		:BOOL			:= FALSE;
	HBcase			:INT			:= 0;
	
   (* received message *)
    SubMCTR		    :BOOL;
	SubIBuff		:BOOL;
    SubHB			:BOOL;
    {attribute 'TcEncoding':='UTF-8'}
    sTopicRcv       :STRING(255);
    {attribute 'TcEncoding':='UTF-8'}
    sPayloadRcv     :STRING(2000);
    fbMessageQueue  :FB_IotMqttMessageQueue;
    fbMessage       :FB_IotMqttMessage;	
	
	(* JSON *)
	fbJson 			:FB_JsonSaxWriter;
	fbJsonDataType 	:FB_JsonReadWriteDataType;
	fbJsonSaxReader	:FB_JsonSaxReader;
	pJsonParse		:JsonSaxHandler;
	jsonDoc    		:SJsonValue;
  	jsonProp   		:SJsonValue;
	
	ok				:BOOL;
	error			:HRESULT;
	index			:INT			:= 0;
	payload			:T_MaxString;
	scriptcnt		:INT			:= 0;
END_VAR

//takes any INT as UDINT?
//received (and echoed) messages:
//GVL_MOTION.EXT_CTR
//GVL_MOTION.InstructionBuffer
//published messages:
//GVL_MOTION.STATUS
//receive 
//GVL_MOTION.HB.HEARTBEAT

IF bSetParameter THEN
    bSetParameter								:= FALSE;
    fbMqttClient.sHostName						:= '127.0.0.1';
    fbMqttClient.nHostPort						:= 1883;
    fbMqttClient.ipMessageQueue					:= fbMessageQueue;
END_IF

fbMqttClient.Execute(bConnect);

IF fbMessageQueue.nQueuedMessages > 0 THEN
    IF fbMessageQueue.Dequeue(fbMessage:=fbMessage) THEN
        fbMessage.GetTopic(pTopic:=ADR(GVL_MOTION.TopicRcv), nTopicSize:=SIZEOF(GVL_MOTION.TopicRcv) );
        fbMessage.GetPayload(pPayload:=ADR(sPayloadRcv), nPayloadSize:=SIZEOF(sPayloadRcv), bSetNullTermination:=FALSE);
		fbJsonSaxReader.Parse(sJson := sPayloadRcv, ipHdl := pJsonParse);
		
    END_IF
END_IF

IF fbMqttClient.bConnected THEN
    IF NOT SubMCTR THEN
        SubMCTR := fbMqttClient.Subscribe(sTopic:='MOTION/CTR', eQoS:=TcIotMqttQos.AtMostOnceDelivery);
    END_IF
    IF NOT SubIBuff THEN
        SubIBuff := fbMqttClient.Subscribe(sTopic:='MOTION/INSTR_BUFFER', eQoS:=TcIotMqttQos.AtMostOnceDelivery);
    END_IF	
	IF NOT SubHB THEN
        SubHB := fbMqttClient.Subscribe(sTopic:='MOTION/HB', eQoS:=TcIotMqttQos.AtMostOnceDelivery);
    END_IF	
    fbTimer(IN:=TRUE);
	//wait for trigger from daqtask - instantaneous data ready to transmit
// 	IF GVL_DAQ.DREADY THEN
// 		GVL_DAQ.DREADY			:= FALSE;
// 		fbJson.ResetDocument();
// 		fbJson.StartObject();	
// 		fbJsonDataType.AddJsonKeyValueFromSymbol(fbJson, '', 'DATA', SIZEOF(GVL_DAQ.DATA), ADR(GVL_DAQ.DATA));
// 		fbJson.EndObject();
// 		fbJson.CopyDocument(sPayloadPub, SIZEOF(sPayLoadPub));
// 		
// 		found	:= FIND2(ADR(sPayLoadPub), ADR('}}'));
// 		DELETE2(ADR(sPayLoadPub), ADR(sPayLoadPub), SIZEOF(sPayLoadPub), 1, found + 1);
// 		DELETE2(ADR(sPayLoadPub), ADR(sPayLoadPub), SIZEOF(sPayLoadPub), 4, 1);
// 		
// 		fbMqttClient.Publish(sTopic:= DaqDataPub, pPayload:= ADR(sPayloadPub), 
// 			nPayloadSize:= LEN2(ADR(sPayloadPub)), eQoS:= TcIotMqttQos.AtMostOnceDelivery, 
// 			bRetain:= TRUE, bQueue:= FALSE );	
// 	END_IF
	
    IF fbTimer.Q THEN // publish new payload every second
		//convert xOut to JSON
        fbTimer(IN:=FALSE);
		
		fbJson.ResetDocument();
		fbJson.StartObject();
		//AddJsonValueFromSymbol does not auto format in mosquitto, this one does
		//this function doesnt work with custom data types in the struct
		//3rd variable is the struct type
		fbJsonDataType.AddJsonKeyValueFromSymbol(fbJson, '', 'STATUS', SIZEOF(GVL_MOTION.STATUS), ADR(GVL_MOTION.STATUS));
		//fbJson.AddKeyBool('EN',GVL_MOTION.xCon.Enable);
		fbJson.EndObject();
		fbJson.CopyDocument(sPayloadPub, SIZEOF(sPayLoadPub));
		
		found	:= FIND2(ADR(sPayLoadPub), ADR('}}'));
		DELETE2(ADR(sPayLoadPub), ADR(sPayLoadPub), SIZEOF(sPayLoadPub), 1, found + 1);
		DELETE2(ADR(sPayLoadPub), ADR(sPayLoadPub), SIZEOF(sPayLoadPub), 4, 1);
		
        fbMqttClient.Publish(sTopic:= MotionStatusPub, pPayload:= ADR(sPayloadPub), 
			nPayloadSize:= LEN2(ADR(sPayloadPub)), eQoS:= TcIotMqttQos.AtMostOnceDelivery, 
			bRetain:= TRUE, bQueue:= FALSE );
			
			
		fbJson.ResetDocument();
		fbJson.StartObject();
		fbJsonDataType.AddJsonKeyValueFromSymbol(fbJson, '', 'MOTION_CTR', SIZEOF(GVL_MOTION.EXT_CTR), ADR(GVL_MOTION.EXT_CTR));
		fbJson.EndObject();
		fbJson.CopyDocument(sPayloadPub, SIZEOF(sPayLoadPub));
		
		found	:= FIND2(ADR(sPayLoadPub), ADR('}}'));
		DELETE2(ADR(sPayLoadPub), ADR(sPayLoadPub), SIZEOF(sPayLoadPub), 1, found + 1);
		DELETE2(ADR(sPayLoadPub), ADR(sPayLoadPub), SIZEOF(sPayLoadPub), 4, 1);
		
		fbMqttClient.Publish(sTopic:= MotionCTREcho, pPayload:= ADR(sPayloadPub), 
			nPayloadSize:= LEN2(ADR(sPayloadPub)), eQoS:= TcIotMqttQos.AtMostOnceDelivery, 
			bRetain:= TRUE, bQueue:= FALSE );
		
		fbJson.ResetDocument();
		fbJson.StartObject();	
		fbJsonDataType.AddJsonKeyValueFromSymbol(fbJson, '', 'MOTION_INSTRUCTION', SIZEOF(GVL_MOTION.InstructionBuffer), ADR(GVL_MOTION.InstructionBuffer));
		fbJson.EndObject();
		fbJson.CopyDocument(sPayloadPub, SIZEOF(sPayLoadPub));
		
		found	:= FIND2(ADR(sPayLoadPub), ADR('}}'));
		DELETE2(ADR(sPayLoadPub), ADR(sPayLoadPub), SIZEOF(sPayLoadPub), 1, found + 1);
		DELETE2(ADR(sPayLoadPub), ADR(sPayLoadPub), SIZEOF(sPayLoadPub), 4, 1);
		
		fbMqttClient.Publish(sTopic:= MotionINSTREcho, pPayload:= ADR(sPayloadPub), 
			nPayloadSize:= LEN2(ADR(sPayloadPub)), eQoS:= TcIotMqttQos.AtMostOnceDelivery, 
			bRetain:= TRUE, bQueue:= FALSE );
	
			
		IF GVL_MOTION.LISTSTART THEN
			IF index < GVL_MOTION.LISTCNT THEN
				IF index = 0 THEN
					GVL_MOTION.SCRIPTNAME.start	:= TRUE;
				ELSIF index = (GVL_MOTION.LISTCNT - 1) THEN
					GVL_MOTION.SCRIPTNAME.end	:= TRUE; 	
				ELSE
					GVL_MOTION.SCRIPTNAME.start	:= FALSE;
					GVL_MOTION.SCRIPTNAME.end	:= FALSE;	
				END_IF
				
				GVL_MOTION.SCRIPTNAME.payload	:= GVL_MOTION.LIST[index];
				
				fbJson.ResetDocument();
				fbJson.StartObject();	
				fbJsonDataType.AddJsonKeyValueFromSymbol(fbJson, '', 'SCRIPTNAME', SIZEOF(GVL_MOTION.SCRIPTNAME), ADR(GVL_MOTION.SCRIPTNAME));
				fbJson.EndObject();
				fbJson.CopyDocument(sPayloadPub, SIZEOF(sPayLoadPub));
				
				found	:= FIND2(ADR(sPayLoadPub), ADR('}}'));
				DELETE2(ADR(sPayLoadPub), ADR(sPayLoadPub), SIZEOF(sPayLoadPub), 1, found + 1);
				DELETE2(ADR(sPayLoadPub), ADR(sPayLoadPub), SIZEOF(sPayLoadPub), 4, 1);
				
				fbMqttClient.Publish(sTopic:= ScriptNames, pPayload:= ADR(sPayloadPub), 
					nPayloadSize:= LEN2(ADR(sPayloadPub)), eQoS:= TcIotMqttQos.AtMostOnceDelivery, 
					bRetain:= TRUE, bQueue:= FALSE );	
					
				index							:= index + 1;
			ELSE
				GVL_MOTION.SCRIPTNAME.start		:= FALSE;
				GVL_MOTION.SCRIPTNAME.end		:= FALSE;
				index							:= 0;	
				GVL_MOTION.LISTSTART			:= FALSE;
				GVL_MOTION.LISTEND				:= TRUE;
			END_IF
		END_IF
    END_IF
END_IF

IF fbMqttClient.bConnected THEN
	//IF GVL_MOTION.EXT_CTR.CMDREQSCRIPT THEN
		scriptTimer(IN:=TRUE);
		IF scriptTimer.Q THEN
			scriptTimer(IN:=FALSE);
			IF scriptcnt < GVL_MOTION.STATUS.ScriptEnd THEN
				GVL_MOTION.Script[scriptcnt].index	:= scriptcnt;
				fbJson.ResetDocument();
				fbJson.StartObject();	
				fbJsonDataType.AddJsonKeyValueFromSymbol(fbJson, '', 'MOTION_INSTRUCTION', SIZEOF(GVL_MOTION.Script[scriptcnt]), ADR(GVL_MOTION.Script[scriptcnt]));
				fbJson.EndObject();
				fbJson.CopyDocument(sPayloadPub, SIZEOF(sPayLoadPub));
				
				found	:= FIND2(ADR(sPayLoadPub), ADR('}}'));
				DELETE2(ADR(sPayLoadPub), ADR(sPayLoadPub), SIZEOF(sPayLoadPub), 1, found + 1);
				DELETE2(ADR(sPayLoadPub), ADR(sPayLoadPub), SIZEOF(sPayLoadPub), 4, 1);
				
				fbMqttClient.Publish(sTopic:= ScriptSend, pPayload:= ADR(sPayloadPub), 
					nPayloadSize:= LEN2(ADR(sPayloadPub)), eQoS:= TcIotMqttQos.AtMostOnceDelivery, 
					bRetain:= TRUE, bQueue:= FALSE );
				scriptcnt						:= scriptcnt + 1;
			ELSE
				scriptcnt						:= 0;
				GVL_MOTION.EXT_CTR.CMDREQSCRIPT	:= FALSE;
			END_IF
		END_IF
	//END_IF
END_IF

IF NOT GVL_MOTION.HB.HEARTBEAT THEN
//3 second timer. set heartbeat false. control continuously sets heartbeat true, 
//after 3 cycles disable sensitive motion controls
	HBtimer(IN:=TRUE, PT := T#1S); 
ELSE
	HBtimer(IN:=FALSE);
	GVL_MOTION.HB.HEARTBEAT						:= FALSE;
END_IF	

IF HBtimer.Q THEN	
	GVL_MOTION.EXT_CTR.XJOGFW					:= FALSE;	
	GVL_MOTION.EXT_CTR.XJOGBW					:= FALSE;	
	GVL_MOTION.EXT_CTR.YJOGFW					:= FALSE;	
	GVL_MOTION.EXT_CTR.YJOGBW					:= FALSE;	
	GVL_MOTION.EXT_CTR.ZJOGFW					:= FALSE;	
	GVL_MOTION.EXT_CTR.ZJOGBW					:= FALSE;	
END_IF

END_PROGRAM

// ---- POUs/JsonSaxHandler.TcPOU
{attribute 'c++_compatible'}
FUNCTION_BLOCK JsonSaxHandler IMPLEMENTS ITcJsonSaxHandler
VAR_INPUT
END_VAR
VAR_OUTPUT
END_VAR
VAR
	(* Values from JSON - written by callback methods *)	  
	keystate			: INT := 0;
	label				: STRING(255);
	tempkey				: STRING(255);
	
	(* State machine variables *)
	//eState				: E_JsonStates;
	
	(* Indicators if an expected property has been found in JSON *)
	bStartObjectFound 	: BOOL;
	bEndObjectFound		: BOOL;
	
	(* Error indicators *)
	bError				: BOOL;
	sErrorMsg			: STRING(255);
END_VAR

IF bError THEN
	sErrorMsg := 'JSON message does not equal expected format';
END_IF

{attribute 'show'}
{attribute 'c++_compatible'}
{attribute 'minimal_input_size' := '4'}
{attribute 'pack_mode' := '4'}
METHOD OnBool : HRESULT
VAR_INPUT
	value	: BOOL;
END_VAR

	IF label = 'MOTION/CTR' THEN
		IF tempkey = 'CMDADD' THEN
			GVL_MOTION.EXT_CTR.CMDADD := value;
		ELSIF tempkey = 'CMDCLR' THEN
			GVL_MOTION.EXT_CTR.CMDCLR := value;
		ELSIF tempkey = 'CMDSCRIPTDEL' THEN
			GVL_MOTION.EXT_CTR.CMDSCRIPTDEL := value;	
		ELSIF tempkey = 'CMDDEL' THEN
			GVL_MOTION.EXT_CTR.CMDDEL := value;	
		ELSIF tempkey = 'CMDRUN' THEN
			GVL_MOTION.EXT_CTR.CMDRUN := value;
		ELSIF tempkey = 'CMDLOOP' THEN
			GVL_MOTION.EXT_CTR.CMDLOOP := value;	
		ELSIF tempkey = 'CMDHOME' THEN
			GVL_MOTION.EXT_CTR.CMDHOME := value;
		ELSIF tempkey = 'CMDHOMEX' THEN
			GVL_MOTION.EXT_CTR.CMDHOMEX := value;
		ELSIF tempkey = 'CMDHOMEY' THEN
			GVL_MOTION.EXT_CTR.CMDHOMEY := value;
		ELSIF tempkey = 'CMDHOMEZ' THEN
			GVL_MOTION.EXT_CTR.CMDHOMEZ := value;	
		ELSIF tempkey = 'CMDCOUPLE' THEN
			GVL_MOTION.EXT_CTR.CMDCOUPLE := value;				
		ELSIF tempkey = 'CMDLOOP' THEN
			GVL_MOTION.EXT_CTR.CMDLOOP := value;	
		ELSIF tempkey = 'STOP' THEN
			GVL_MOTION.EXT_CTR.STOP := value;	
		ELSIF tempkey = 'AXESEN' THEN
			GVL_MOTION.EXT_CTR.AXESEN := value;		
		ELSIF tempkey = 'AXESRESET' THEN
			GVL_MOTION.EXT_CTR.AXESRESET := value;	
		ELSIF tempkey = 'CMDSCRIPTWRITE' THEN
			GVL_MOTION.EXT_CTR.CMDSCRIPTWRITE := value;
		ELSIF tempkey = 'CMDSCRIPTREAD' THEN
			GVL_MOTION.EXT_CTR.CMDSCRIPTREAD := value;	
		ELSIF tempkey = 'CMDREQLIST' THEN
			GVL_MOTION.EXT_CTR.CMDREQLIST := value;
		ELSIF tempkey = 'CMDREQSCRIPT' THEN
			GVL_MOTION.EXT_CTR.CMDREQSCRIPT := value;	
		ELSIF tempkey = 'XJOGFW' THEN
			GVL_MOTION.EXT_CTR.XJOGFW := value;
		ELSIF tempkey = 'XJOGBW' THEN
			GVL_MOTION.EXT_CTR.XJOGBW := value;
		ELSIF tempkey = 'YJOGFW' THEN
			GVL_MOTION.EXT_CTR.YJOGFW := value;
		ELSIF tempkey = 'YJOGBW' THEN
			GVL_MOTION.EXT_CTR.YJOGBW := value;
		ELSIF tempkey = 'ZJOGFW' THEN
			GVL_MOTION.EXT_CTR.ZJOGFW := value;
		ELSIF tempkey = 'ZJOGBW' THEN
			GVL_MOTION.EXT_CTR.ZJOGBW := value;	
		ELSIF tempkey = 'SETXPOS' THEN
			GVL_MOTION.EXT_CTR.SETXPOS := value;
		ELSIF tempkey = 'SETYPOS' THEN
			GVL_MOTION.EXT_CTR.SETYPOS := value;
		ELSIF tempkey = 'SETZPOS' THEN
			GVL_MOTION.EXT_CTR.SETZPOS := value;	
		ELSIF tempkey = 'BASINCTR' THEN
			GVL_MOTION.EXT_CTR.BASINCTR := value;
		ELSIF tempkey = 'BRAKEREL' THEN
			GVL_MOTION.EXT_CTR.BRAKEREL := value;
		ELSIF tempkey = 'MOVEX' THEN
			GVL_MOTION.EXT_CTR.MOVEX := value;
		ELSIF tempkey = 'MOVEY' THEN
			GVL_MOTION.EXT_CTR.MOVEY := value;
		ELSIF tempkey = 'MOVEZ' THEN
			GVL_MOTION.EXT_CTR.MOVEZ := value;							
		END_IF		
	ELSIF label = 'MOTION/HB' THEN
		IF tempkey = 'HEARTBEAT' THEN
			GVL_MOTION.HB.HEARTBEAT := value;
		END_IF	
// 	ELSIF label = 'DAQ/CTR' THEN
// 		IF tempkey = 'CMDDATACLR' THEN
// 			GVL_DAQ.TEST_CTR.CMDDATACLR := value;	
// 		ELSIF tempkey = 'CMDDATAAPEND' THEN
// 			GVL_DAQ.TEST_CTR.CMDDATAAPEND := value;
// 		ELSIF tempkey = 'CMDDATAWRITE' THEN
// 			GVL_DAQ.TEST_CTR.CMDDATAWRITE := value;
// 		END_IF	
// 	ELSIF label = 'MOTION/INSTR_BUFFER' THEN
// 		IF tempkey = 'Acq_Keyence' THEN
// 			GVL_MOTION.TestBuffer.Acq_Keyence := value;
// 		ELSIF tempkey = 'Acq_Massa' THEN
// 			GVL_MOTION.TestBuffer.Acq_Massa := value;
// 		ELSIF tempkey = 'Acq_Sonar' THEN
// 			GVL_MOTION.TestBuffer.Acq_Sonar := value;
// 		END_IF	
		
	END_IF
END_METHOD

{attribute 'show'}
{attribute 'c++_compatible'}
{attribute 'minimal_input_size' := '4'}
{attribute 'pack_mode' := '4'}
METHOD OnDint : HRESULT
VAR_INPUT
	value	: DINT;
END_VAR
// := value;
END_METHOD

{attribute 'show'}
{attribute 'c++_compatible'}
{attribute 'minimal_input_size' := '4'}
{attribute 'pack_mode' := '4'}
METHOD OnEndArray : HRESULT
VAR_INPUT
	elementCount	: UDINT;
END_VAR
END_METHOD

{attribute 'show'}
{attribute 'c++_compatible'}
{attribute 'minimal_input_size' := '4'}
{attribute 'pack_mode' := '4'}
METHOD OnEndObject : HRESULT
VAR_INPUT
	memberCount	: UDINT;
END_VAR
// IF (eState = 100) THEN
// 	bEndObjectFound := TRUE;
// 	eState := 110;  
// 	ELSE
// 		IF (eState = 110) THEN
// 			bEndObjectFound := TRUE;
// 			eState := 120;
// 		ELSE
// 			bError := TRUE;  
// 	  END_IF			
// END_IF

//keystate := keystate - 1;
END_METHOD

{attribute 'show'}
{attribute 'c++_compatible'}
{attribute 'minimal_input_size' := '4'}
{attribute 'pack_mode' := '4'}
METHOD OnKey : HRESULT
VAR_IN_OUT CONSTANT
	key	: STRING;
END_VAR
VAR_INPUT
	len	: UDINT;
END_VAR


// IF keystate = 1 THEN
// 	label := key;
// ELSIF keystate > 1 THEN
// 	tempkey	:= key;
// 	bStartObjectFound := FALSE;
// END_IF

tempkey	:= key;
END_METHOD

{attribute 'show'}
{attribute 'c++_compatible'}
{attribute 'minimal_input_size' := '4'}
{attribute 'pack_mode' := '4'}
METHOD OnLint : HRESULT
VAR_INPUT
	value	: LINT;
END_VAR
END_METHOD

{attribute 'show'}
{attribute 'c++_compatible'}
{attribute 'minimal_input_size' := '4'}
{attribute 'pack_mode' := '4'}
METHOD OnLreal : HRESULT
VAR_INPUT
	value	: LREAL;
END_VAR
// IF (eState = 70) THEN
// 	bSensor1ValueFound := TRUE;
// 	Sensor1 := value;
// 	eState := 80;
// ELSE
// 	bError := TRUE;
// 	OnLreal := S_FALSE;
// END_IF

	IF label = 'MOTION/INSTR_BUFFER' THEN
		IF tempkey = 'SetXPosition' THEN
			GVL_MOTION.InstructionBuffer.SetXPosition		:= value;
		ELSIF tempkey = 'SetYPosition' THEN
			GVL_MOTION.InstructionBuffer.SetYPosition		:= value;
		ELSIF tempkey = 'SetZPosition' THEN
			GVL_MOTION.InstructionBuffer.SetZPosition		:= value;	
		END_IF
	ELSIF label = 'MOTION/CTR' THEN	
		IF tempkey = 'POSX' THEN
			GVL_MOTION.EXT_CTR.POSX		:= value;
		ELSIF tempkey = 'POSY' THEN
			GVL_MOTION.EXT_CTR.POSY		:= value;
		ELSIF tempkey = 'POSZ' THEN
			GVL_MOTION.EXT_CTR.POSZ		:= value;	
		END_IF
	END_IF
END_METHOD

{attribute 'show'}
{attribute 'c++_compatible'}
{attribute 'minimal_input_size' := '4'}
{attribute 'pack_mode' := '4'}
METHOD OnNull : HRESULT
END_METHOD

{attribute 'show'}
{attribute 'c++_compatible'}
{attribute 'minimal_input_size' := '4'}
{attribute 'pack_mode' := '4'}
METHOD OnRawNumber : HRESULT
VAR_IN_OUT CONSTANT
	value	: STRING;
END_VAR
VAR_INPUT
	len	: UDINT;
END_VAR
END_METHOD

{attribute 'show'}
{attribute 'c++_compatible'}
{attribute 'minimal_input_size' := '4'}
{attribute 'pack_mode' := '4'}
METHOD OnStartArray : HRESULT
END_METHOD

{attribute 'show'}
{attribute 'c++_compatible'}
{attribute 'minimal_input_size' := '4'}
{attribute 'pack_mode' := '4'}
METHOD OnStartObject : HRESULT

//keystate := keystate + 1;
label := GVL_MOTION.TopicRcv;
bStartObjectFound := TRUE;
END_METHOD

{attribute 'show'}
{attribute 'c++_compatible'}
{attribute 'minimal_input_size' := '4'}
{attribute 'pack_mode' := '4'}
METHOD OnString : HRESULT
VAR_IN_OUT CONSTANT
	value	: STRING;
END_VAR
VAR_INPUT
	len	: UDINT;
END_VAR
// IF (eState = 50) THEN
// 	bTimestampValueFound := TRUE;
// 	STRNCPY(pDst:=ADR(sTimestamp), pSrc:=ADR(value), nDstSize:=SIZEOF(sTimestamp));
// 	eState := 60;
// ELSE
// 	bError := TRUE;
// 	OnString := S_FALSE;
// END_IF

	IF label = 'MOTION/INSTR_BUFFER' THEN
		IF tempkey = 'Comment' THEN
			GVL_MOTION.InstructionBuffer.Comment		:= value;
		END_IF
	ELSIF label = 'MOTION/CTR' THEN
		IF tempkey = 'SCRIPTNAME' THEN
			GVL_MOTION.EXT_CTR.SCRIPTNAME		:= value;
		END_IF	
	END_IF
END_METHOD

{attribute 'show'}
{attribute 'c++_compatible'}
{attribute 'minimal_input_size' := '4'}
{attribute 'pack_mode' := '4'}
METHOD OnUdint : HRESULT
VAR_INPUT
	value		:UDINT;
END_VAR
VAR
	//temptime	:TIME;
END_VAR
// IF (eState = 90) THEN
// 	bSensor2ValueFound := TRUE;
// 	Sensor2 := value;
// 	eState := 100;
// ELSE
// 	bError := TRUE;TO_TIME
// 	OnUdint := S_FALSE;
// END_IF

	IF label = 'MOTION/INSTR_BUFFER' THEN
		IF tempkey = 'MotionCommand' THEN
			GVL_MOTION.InstructionBuffer.MotionCommand		:= UDINT_TO_INT(value);
// 		ELSIF tempkey = 'zType' THEN
// 			GVL_MOTION.TestBuffer.zType				:= UDINT_TO_INT(value);
// 		ELSIF tempkey = 'DataTrigger' THEN
// 			GVL_MOTION.TestBuffer.DataTrigger		:= UDINT_TO_INT(value);	
		ELSIF tempkey = 'SetXPosition' THEN
			GVL_MOTION.InstructionBuffer.SetXPosition		:= UDINT_TO_INT(value);
		ELSIF tempkey = 'SetXVelocity' THEN
			GVL_MOTION.InstructionBuffer.SetXVelocity		:= UDINT_TO_INT(value);
		ELSIF tempkey = 'SetXAccel' THEN
			GVL_MOTION.InstructionBuffer.SetXAccel			:= UDINT_TO_INT(value);
		ELSIF tempkey = 'SetYPosition' THEN
			GVL_MOTION.InstructionBuffer.SetYPosition		:= UDINT_TO_INT(value);
		ELSIF tempkey = 'SetYVelocity' THEN
			GVL_MOTION.InstructionBuffer.SetYVelocity		:= UDINT_TO_INT(value);
		ELSIF tempkey = 'SetYAccel' THEN
			GVL_MOTION.InstructionBuffer.SetYAccel			:= UDINT_TO_INT(value);
		ELSIF tempkey = 'SetZPosition' THEN
			GVL_MOTION.InstructionBuffer.SetZPosition		:= UDINT_TO_INT(value);
		ELSIF tempkey = 'SetZVelocity' THEN
			GVL_MOTION.InstructionBuffer.SetZVelocity		:= UDINT_TO_INT(value);			
		ELSIF tempkey = 'PauseTime' THEN
			//temptime := TIME#1MS * value;
			GVL_MOTION.InstructionBuffer.PauseTime 		:= TIME#1MS * value;
		END_IF		
// 	ELSIF label = 'DAQ/CTR' THEN
// 		IF tempkey = 'DAQRES' THEN
// 			GVL_DAQ.TEST_CTR.DAQRES				:= UDINT_TO_INT(value);
// 		END_IF	
	ELSIF label = 'MOTION/CTR' THEN	
		IF tempkey = 'SCRIPTITERATIONS' THEN 	
			GVL_MOTION.EXT_CTR.SCRIPTITERATIONS	:= UDINT_TO_INT(value);	
		END_IF
		
	END_IF
END_METHOD

{attribute 'show'}
{attribute 'c++_compatible'}
{attribute 'minimal_input_size' := '4'}
{attribute 'pack_mode' := '4'}
METHOD OnUlint : HRESULT
VAR_INPUT
	value	: ULINT;
END_VAR
END_METHOD

{attribute 'show'}
{attribute 'c++_compatible'}
{attribute 'minimal_input_size' := '4'}
{attribute 'pack_mode' := '4'}
METHOD TcAddRef : UDINT
END_METHOD

{attribute 'show'}
{attribute 'c++_compatible'}
{attribute 'minimal_input_size' := '4'}
{attribute 'pack_mode' := '4'}
METHOD TcQueryInterface : HRESULT
VAR_INPUT
	iid	: REFERENCE TO IID;
	pipItf	: POINTER TO PVOID;
END_VAR
END_METHOD

{attribute 'show'}
{attribute 'c++_compatible'}
{attribute 'minimal_input_size' := '4'}
{attribute 'pack_mode' := '4'}
METHOD TcRelease : UDINT
END_METHOD

END_FUNCTION_BLOCK

// ---- POUs/ResetAxes.TcPOU
PROGRAM ResetAxes
VAR
	resetstate				:INT	:= 0;
END_VAR

CASE resetstate OF
	0:
	IF GVL_MOTION.EXT_CTR.AxesReset THEN
		GVL_MOTION.EXT_CTR.AxesReset		:= FALSE;
		GVL_MOTION.HomingState				:= 0;
		GVL_MOTION.xCon.Execute_MREL		:= FALSE;
		//GVL_MOTION.HardStopState			:= 0;
		GVL_MOTION.xCon.Execute_HOME		:= FALSE;
		GVL_MOTION.xcCon.Execute_HOME		:= FALSE;
		GVL_MOTION.xCon.Execute_HALT		:= FALSE;
		GVL_MOTION.xcCon.Execute_HALT		:= FALSE;
		GVL_MOTION.xCon.Execute_RES 		:= TRUE;
		IF NOT GVL_MOTION.xOut.AxisCoupled THEN
			GVL_MOTION.xcCon.Execute_RES	:= TRUE;
		END_IF
		GVL_MOTION.yCon.Execute_HOME		:= FALSE;
		GVL_MOTION.yCon.Execute_HALT		:= FALSE;
		GVL_MOTION.yCon.Execute_RES 		:= TRUE;
		GVL_MOTION.zCon.Execute_HOME		:= FALSE;
		GVL_MOTION.zCon.Execute_HALT		:= FALSE;
		GVL_MOTION.zCon.Execute_RES 		:= TRUE;
		resetstate							:= 1;
	END_IF	
	1:
		GVL_MOTION.xCon.Execute_RES 		:= FALSE;
		GVL_MOTION.xcCon.Execute_RES		:= FALSE;
		GVL_MOTION.yCon.Execute_RES 		:= FALSE;
		GVL_MOTION.zCon.Execute_RES 		:= FALSE;
		resetstate							:= 0;
END_CASE

END_PROGRAM

// ---- POUs/zAxisMoreLogic.TcPOU
PROGRAM zAxisMoreLogic
VAR
	zHaltMem		:BOOL	:= FALSE;
END_VAR

//stop z from slamming into frame
IF GVL_MOTION.zCon.LimNeg AND NOT GVL_MOTION.zCon.Execute_HOME AND NOT zHaltMem AND NOT GVL_MOTION.zSafeDisable THEN
	zHaltMem								:= TRUE;
	GVL_MOTION.zCon.Execute_HALT			:= TRUE;
END_IF

//rearm z safety
IF NOT GVL_MOTION.zCon.LimNeg AND zHaltMem THEN
	GVL_MOTION.zCon.Execute_HALT			:= FALSE;
	zHaltMem								:= FALSE;
END_IF

END_PROGRAM

// ---- POUs/ScriptList.TcPOU
PROGRAM ScriptList
VAR
	fbEnum: FB_EnumFindFileEntry := ( sNetID := '', tTimeout := T#5S, sPathName := 'C:\MOTION_SCRIPTS\*.csv' );
    bEnum	:BOOL;
    bAbort	:BOOL;
    nState	:BYTE;
	found	:UDINT;
END_VAR

CASE nState OF
    0:
		//if requestlist
        IF GVL_MOTION.EXT_CTR.CMDREQLIST THEN             (* flag set ? *)
            GVL_MOTION.EXT_CTR.CMDREQLIST						:= FALSE;         (* reset flag *)
			
            fbEnum.eCmd := eEnumCmd_First;    (* enum first entry *)
            nState												:= 1;
        END_IF

    1:    (* enum one entry *)
        IF bAbort THEN
            bAbort												:= FALSE;
            fbEnum.eCmd											:= eEnumCmd_Abort;
        END_IF
        fbEnum( bExecute := FALSE );
        fbEnum( bExecute := TRUE );
        nState													:= 2;

    2:    (* wait until function block not busy *)
        fbEnum( bExecute := FALSE );
        IF NOT fbEnum.bBusy THEN
            IF NOT fbEnum.bError THEN
                IF NOT fbEnum.bEOE THEN
						IF GVL_MOTION.LISTCNT < 1000 THEN
						GVL_MOTION.LIST[GVL_MOTION.LISTCNT]		:= fbEnum.stFindFile.sFileName;
						found									:= FIND2(ADR(GVL_MOTION.LIST[GVL_MOTION.LISTCNT]), ADR('_Script.csv'));
						IF found <> 0 THEN
							//delete '_Script.csv' from title
							DELETE2(ADR(GVL_MOTION.LIST[GVL_MOTION.LISTCNT])
								   ,ADR(GVL_MOTION.LIST[GVL_MOTION.LISTCNT])
								   ,SIZEOF(GVL_MOTION.LIST[GVL_MOTION.LISTCNT])
								   ,11
								   ,found);
							GVL_MOTION.LISTCNT		:= GVL_MOTION.LISTCNT + 1;
						END_IF
						fbEnum.eCmd := eEnumCmd_Next; (* enum next entry *)
						nState      := 1;
						ELSE
							GVL_MOTION.STATUS.List_Overflow_Err	:= TRUE;
							GVL_MOTION.LISTCNT					:= 0;
							nState								:= 0;
						END_IF	
                ELSE (* no more entries *)
					//GVL_MOTION.LISTCNT	:= 1;
					GVL_MOTION.LISTSTART						:= TRUE;
                    nState     									:= 3;
                END_IF
            ELSE (* log error *)
                ADSLOGSTR( ADSLOG_MSGTYPE_ERROR OR ADSLOG_MSGTYPE_LOG, 'FB_EnumFindFileEntry error:%s', DWORD_TO_HEXSTR( fbEnum.nErrID, 0, FALSE ) );
                nState    										:= 0;
            END_IF
        END_IF
	3:
		//wait for LISTDONE and reset variables
		IF GVL_MOTION.LISTEND THEN
			GVL_MOTION.LISTCNT									:= 0;
			nState												:= 0;
			GVL_MOTION.LISTEND									:= FALSE;
		END_IF
END_CASE

END_PROGRAM

// ---- POUs/DeleteScriptFile.TcPOU
PROGRAM DeleteScriptFile
VAR
	step			:INT	:= 0;
	directory		:T_MaxString	:= 'C:\MOTION_SCRIPTS';
	CMDPATH			:T_MaxString	:= 'C:\Windows\System32\cmd.exe';
	COMNDLINE		:T_MaxString	:= '/C "del '; // /C carries out command string then terminates
	fbCMD			:NT_StartProcess; //run CMD to create data directories
END_VAR

CASE step OF
	0:
	IF GVL_MOTION.EXT_CTR.CMDSCRIPTDEL THEN
		GVL_MOTION.EXT_CTR.CMDSCRIPTDEL	:= FALSE;
		COMNDLINE						:= concat('/C "del ', GVL_MOTION.EXT_CTR.SCRIPTNAME);
		COMNDLINE						:= concat(COMNDLINE, '_Script.csv');
		step							:= 1;
	END_IF
	
	1:
		fbCMD( PATHSTR:= CMDPATH, DIRNAME:= directory, COMNDLINE:= COMNDLINE, START:= TRUE);
		fbCMD(START:= FALSE);
		IF NOT fbCMD.BUSY THEN
			step 						:= 0;
		END_IF
END_CASE

END_PROGRAM

// ---- POUs/HomeX.TcPOU
PROGRAM HomeX
VAR
	state		:INT	:= 99;
END_VAR

IF GVL_MOTION.EXT_CTR.CMDHOMEX THEN
	GVL_MOTION.EXT_CTR.CMDHOMEX				:= FALSE;
	GVL_MOTION.xCon.IsHoming				:= TRUE;
	state									:= 0;
END_IF

CASE state OF
	0:
	IF NOT GVL_MOTION.xOut.AxisCoupled THEN
		GVL_MOTION.xCon.ExecuteUncouple		:= FALSE;
		GVL_MOTION.xCon.ExecuteCouple		:= TRUE;
	END_IF
	state									:= 1;
	
	1:
	IF GVL_MOTION.xOut.AxisCoupled THEN
		GVL_MOTION.xJogBW					:= TRUE;
		state								:= 2;
	END_IF
	
	2:
	IF GVL_MOTION.xCon.LimNeg OR GVL_MOTION.xcCon.LimNeg THEN
		GVL_MOTION.xJogBW					:= FALSE;
		GVL_MOTION.xCon.SetPosition			:= 5;
		GVL_MOTION.xCon.SetVelocity			:= 50;
		
		state								:= 3;
	END_IF
	
	3:
	GVL_MOTION.xCon.Execute_MREL			:= TRUE;
	state									:= 4;

	4:
	IF GVL_MOTION.xOut.MoveDone THEN
		GVL_MOTION.xCon.Execute_MREL		:= FALSE;
		GVL_MOTION.xCon.ExecuteCouple		:= FALSE;
		GVL_MOTION.xCon.ExecuteUncouple 	:= TRUE;
		state								:= 5;
	END_IF
	
	5:
	IF NOT GVL_MOTION.xOut.AxisCoupled THEN
		GVL_MOTION.xCon.Execute_HOME		:= TRUE; 
		state								:= 6;
	END_IF
	
	6:
	IF GVL_MOTION.xHomeStatus.Done THEN
		GVL_MOTION.xCon.Execute_HOME		:= FALSE;
		GVL_MOTION.xcCon.Execute_HOME		:= TRUE;
 		state								:= 7;
	END_IF
	
	7:
	IF GVL_MOTION.xcHomeStatus.Done THEN
		GVL_MOTION.xcCon.Execute_HOME		:= FALSE;
		GVL_MOTION.xCon.ExecuteUncouple 	:= FALSE;
		state								:= 8;
	END_IF
	
	8:
	state									:= 99;
	GVL_MOTION.xCon.ExecuteCouple			:= TRUE;
	GVL_MOTION.xLocated						:= TRUE;
	GVL_MOTION.xCon.IsHoming				:= FALSE;
	
	99:; //idle
END_CASE

END_PROGRAM

// ---- POUs/HomeY.TcPOU
PROGRAM HomeY
VAR
	state	:INT	:= 99;
END_VAR

IF GVL_MOTION.EXT_CTR.CMDHOMEY THEN
	GVL_MOTION.EXT_CTR.CMDHOMEY				:= FALSE;
	GVL_MOTION.yCon.IsHoming				:= TRUE;
	state									:= 0;
END_IF

CASE state OF
	0:
	GVL_MOTION.yCon.Execute_HOME		:= TRUE;
	state								:= 1;
	
	1:
	IF GVL_MOTION.yHomeStatus.Done THEN
		GVL_MOTION.yCon.Execute_HOME	:= FALSE;
		GVL_MOTION.yLocated				:= TRUE;
		state							:= 99;
		GVL_MOTION.yCon.IsHoming		:= FALSE;
	END_IF
	
	99:; //idle
END_CASE

END_PROGRAM

// ---- POUs/HomeZ.TcPOU
PROGRAM HomeZ
VAR
	state	:INT	:= 99;
END_VAR

IF GVL_MOTION.EXT_CTR.CMDHOMEZ THEN
	GVL_MOTION.EXT_CTR.CMDHOMEZ				:= FALSE;
	GVL_MOTION.zCon.IsHoming				:= TRUE;
	state									:= 0;
END_IF

CASE state OF
	0:
	GVL_MOTION.zCon.Execute_HOME		:= TRUE;
	state								:= 1;
	
	1:
	IF GVL_MOTION.zHomeStatus.Done THEN
		GVL_MOTION.zCon.Execute_HOME	:= FALSE;
		GVL_MOTION.zLocated				:= TRUE;
		state							:= 99;
		GVL_MOTION.zCon.IsHoming		:= FALSE;
	END_IF	
	
	99:; //idle

END_CASE

END_PROGRAM

// ---- POUs/AddCommand.TcPOU
PROGRAM AddCommand
VAR
END_VAR

IF GVL_MOTION.EXT_CTR.CMDADD THEN
	GVL_MOTION.EXT_CTR.CMDADD					:= FALSE;
	//QueueEnd contains no data
	IF GVL_MOTION.ScriptEnd < 100 THEN
		GVL_MOTION.Script[GVL_MOTION.ScriptEnd]	:= GVL_MOTION.InstructionBuffer;
		GVL_MOTION.ScriptEnd 					:= GVL_MOTION.ScriptEnd + 1;
		GVL_MOTION.EXT_CTR.CMDADD 				:= FALSE;
	ELSE
		//error msg
		GVL_MOTION.EXT_CTR.CMDADD 				:= FALSE;
	END_IF

END_IF

END_PROGRAM

// ---- POUs/DeleteLastInstruction.TcPOU
PROGRAM DeleteLastInstruction
VAR
END_VAR

IF GVL_MOTION.EXT_CTR.CMDDEL THEN
	GVL_MOTION.EXT_CTR.CMDDEL					:= FALSE;
	//QueueEnd contains no data
	IF GVL_MOTION.ScriptEnd <> 0 THEN
		GVL_MOTION.ScriptEnd 					:= GVL_MOTION.ScriptEnd - 1;
		GVL_MOTION.Script[GVL_MOTION.ScriptEnd]	:= GVL_MOTION.EmptyInstruction;
		GVL_MOTION.EXT_CTR.CMDDEL 				:= FALSE;
	ELSE
		//error msg
		GVL_MOTION.EXT_CTR.CMDDEL 				:= FALSE;
	END_IF

END_IF

END_PROGRAM

// ---- POUs/DirectMotion.TcPOU
PROGRAM DirectMotion
VAR
	state	:INT	:= 0;
	timer	:TON;
	fromX	:BOOL;
	fromY	:BOOL;
	fromZ	:BOOL;
END_VAR

CASE state OF
0:	
	timer(IN:=TRUE,PT:=T#30MS); //debounce
	IF timer.Q THEN
		IF GVL_MOTION.EXT_CTR.MOVEX THEN
			fromX									:= TRUE;
			state									:= 2;
			
		ELSIF GVL_MOTION.EXT_CTR.MOVEY THEN 	
			fromY									:= TRUE;
			state									:= 3;
		
		ELSIF GVL_MOTION.EXT_CTR.MOVEZ THEN 	
			fromZ									:= TRUE;
			state									:= 4;
			
		END_IF	
	END_IF	
	
1:
	GVL_MOTION.xCon.Execute_MABS					:= FALSE;
	GVL_MOTION.yCon.Execute_MABS					:= FALSE;
	GVL_MOTION.zCon.Execute_MABS					:= FALSE;
	GVL_MOTION.xCon.Execute_HALT					:= TRUE;
	GVL_MOTION.yCon.Execute_HALT					:= TRUE;
	GVL_MOTION.zCon.Execute_HALT					:= TRUE;
	timer(IN:=TRUE,PT:=T#30MS);
	IF timer.Q THEN
		IF GVL_MOTION.STOP_INT THEN
			timer(IN:=FALSE);
			GVL_MOTION.xCon.Execute_HALT			:= FALSE;
			GVL_MOTION.yCon.Execute_HALT			:= FALSE;
			GVL_MOTION.zCon.Execute_HALT			:= FALSE;
			IF fromX THEN
				state								:= 2;
			ELSIF fromY THEN
				state								:= 3;
			ELSIF fromZ	THEN
				state								:= 4;	
			END_IF
		END_IF
		
	END_IF
	
2:
	IF  GVL_MOTION.EXT_CTR.POSX < GVL_MOTION.STATUS.HardStopLocations[0]
	AND GVL_MOTION.EXT_CTR.POSX > GVL_MOTION.STATUS.CARRIAGE_OFFSETS[0]
	THEN
		IF GVL_MOTION.STOP_INT THEN
			state									:= 1;
		ELSE
			GVL_MOTION.xCon.SetPosition				:= GVL_MOTION.EXT_CTR.POSX - GVL_MOTION.CARRIAGE_OFFSETS[0];
			GVL_MOTION.xCon.SetVelocity				:= 200;
			GVL_MOTION.xCon.Execute_MABS			:= TRUE;
			
			IF GVL_MOTION.xOut.MoveDone THEN
				GVL_MOTION.xCon.Execute_MABS		:= FALSE;
				fromX								:= FALSE;
				state								:= 0;
			END_IF
		END_IF
	ELSE
		state										:= 0;	
	END_IF	
	
3:
	IF  GVL_MOTION.EXT_CTR.POSY < GVL_MOTION.STATUS.HardStopLocations[1]
	AND GVL_MOTION.EXT_CTR.POSY > GVL_MOTION.STATUS.CARRIAGE_OFFSETS[1]
	THEN
		IF GVL_MOTION.STOP_INT THEN
			state									:= 1;
		ELSE	
			GVL_MOTION.yCon.SetPosition				:= GVL_MOTION.EXT_CTR.POSY - GVL_MOTION.CARRIAGE_OFFSETS[1];
			GVL_MOTION.yCon.SetVelocity				:= 200;
			GVL_MOTION.yCon.Execute_MABS			:= TRUE;
			IF GVL_MOTION.yOut.MoveDone THEN
				GVL_MOTION.yCon.Execute_MABS		:= FALSE;
				fromY								:= FALSE;
				GVL_MOTION.EXT_CTR.MOVEY			:= FALSE;
			END_IF
		END_IF
	ELSE
		state										:= 0;	
	END_IF	

4:
	IF  GVL_MOTION.EXT_CTR.POSZ < GVL_MOTION.STATUS.HardStopLocations[2]
	AND GVL_MOTION.EXT_CTR.POSZ > GVL_MOTION.STATUS.CARRIAGE_OFFSETS[2]
	THEN
		IF GVL_MOTION.STOP_INT THEN
			GVL_MOTION.Z_BRAKE_OFF					:= FALSE;
			state									:= 1;
		ELSE
			GVL_MOTION.Z_BRAKE_OFF					:= TRUE;
			GVL_MOTION.zCon.SetPosition				:= GVL_MOTION.EXT_CTR.POSZ - GVL_MOTION.CARRIAGE_OFFSETS[2];
			GVL_MOTION.zCon.SetVelocity				:= 80;
			GVL_MOTION.zCon.Execute_MABS			:= TRUE;
			IF GVL_MOTION.zOut.MoveDone THEN
				GVL_MOTION.Z_BRAKE_OFF				:= FALSE;
				GVL_MOTION.zCon.Execute_MABS		:= FALSE;
				GVL_MOTION.EXT_CTR.MOVEZ			:= FALSE;
			END_IF
		END_IF
	ELSE
		state										:= 0;	
	END_IF	
	
END_CASE

END_PROGRAM

// ---- POUs/RunCommands.TcPOU
PROGRAM RunCommands
VAR
	timer		:TON;
	t2			:TON;
	t3			:TON;
	t4			:TON;
	t5			:TON;
	hold		:TIME;
	index		:INT;
	(*set to true during daq instruction when future daq instructions are detected. delay daq execution until last daq instruction in script*)
	DAQ_HOLD	:BOOL	:= FALSE;
	dataclr		:BOOL	:= FALSE;
	error		:BOOL	:= FALSE;
	SICK_CPP	:NT_StartProcess; //run SICK_Control CPP 
END_VAR



//script exits: state 0,1,3
CASE GVL_MOTION.InstructionState OF
	//WaitOK command type stays in state 0
	//state 0: set axes destinations and enable/send to state 1 or set data acquistion along single axis and enable/send to state 4
	0:
	GVL_MOTION.STATUS.Move_Rel_Err								:= FALSE;
	GVL_MOTION.STATUS.Move_Abs_Err								:= FALSE;
	//GVL_MOTION.STATUS.HS_Err									:= FALSE;
	GVL_MOTION.STATUS.Basin_Exceed_Err							:= FALSE;
	error														:= FALSE;
	
	IF GVL_MOTION.Script[GVL_MOTION.CurInstruction].MotionCommand = MotionType.WaitOK THEN
		IF NOT GVL_MOTION.HaltMem THEN
			GVL_MOTION.HaltMem 									:= TRUE;
			GVL_MOTION.xCon.Execute_HALT						:= TRUE;
			GVL_MOTION.yCon.Execute_HALT						:= TRUE;
			GVL_MOTION.zCon.Execute_HALT						:= TRUE;
			//GVL_MOTION.EXT_CTR.PAUSE							:= TRUE;
			GVL_MOTION.TxtBxWaitOK								:= FALSE;	
		END_IF
		
		IF GVL_MOTION.STOP_INT THEN
			GVL_MOTION.HaltMem									:= FALSE;
			GVL_MOTION.TxtBxWaitOK								:= TRUE;
			GVL_MOTION.xCon.Execute_HALT						:= FALSE;
			GVL_MOTION.yCon.Execute_HALT						:= FALSE;
			GVL_MOTION.zCon.Execute_HALT						:= FALSE;	
			
			IF GVL_MOTION.CurInstruction < (GVL_MOTION.ScriptEnd - 1) THEN
				GVL_MOTION.CurInstruction 						:= GVL_MOTION.CurInstruction + 1; //queue next instruction
			ELSE
				GVL_MOTION.CurInstruction						:= 0;
				IF NOT GVL_MOTION.EXT_CTR.CMDLOOP THEN
					IF GVL_MOTION.RUN_INDEX >= GVL_MOTION.EXT_CTR.SCRIPTITERATIONS THEN
						GVL_MOTION.RUN_INDEX					:= 1;
						GVL_MOTION.EXT_CTR.CMDRUN 				:= FALSE;	 //command list executed
					ELSE
						GVL_MOTION.RUN_INDEX					:= GVL_MOTION.RUN_INDEX + 1;	
					END_IF
					
				ELSE
					GVL_MOTION.RUN_INDEX						:= GVL_MOTION.RUN_INDEX + 1;
				END_IF
				
			END_IF
			
		END_IF	
		
	ELSIF(GVL_MOTION.Script[GVL_MOTION.CurInstruction].MotionCommand = MotionType.Absolute)
	OR	 (GVL_MOTION.Script[GVL_MOTION.CurInstruction].MotionCommand = MotionType.Relative) 
	THEN
		
		IF GVL_MOTION.Script[GVL_MOTION.CurInstruction].MotionCommand = MotionType.Absolute THEN
			
				//check hard stops
// 				IF ((GVL_MOTION.Script[GVL_MOTION.CurInstruction].SetXPosition < GVL_MOTION.STATUS.HardStopLocations[0])
// 				AND((GVL_MOTION.Script[GVL_MOTION.CurInstruction].SetYPosition < GVL_MOTION.STATUS.HardStopLocations[1])
// 				AND((GVL_MOTION.Script[GVL_MOTION.CurInstruction].SetZPosition < GVL_MOTION.STATUS.HardStopLocations[2])
// 				THEN
				//check basin
				IF  (GVL_MOTION.Script[GVL_MOTION.CurInstruction].SetXPosition > GVL_MOTION.ActiveBasin.xMin)
				AND (GVL_MOTION.Script[GVL_MOTION.CurInstruction].SetXPosition < GVL_MOTION.ActiveBasin.xMax)
				AND (GVL_MOTION.Script[GVL_MOTION.CurInstruction].SetYPosition > GVL_MOTION.ActiveBasin.yMin)
				AND (GVL_MOTION.Script[GVL_MOTION.CurInstruction].SetYPosition < GVL_MOTION.ActiveBasin.yMax)
				AND (GVL_MOTION.Script[GVL_MOTION.CurInstruction].SetZPosition > 0)
				AND (GVL_MOTION.Script[GVL_MOTION.CurInstruction].SetZPosition < GVL_MOTION.STATUS.HardStopLocations[2])
				THEN
					GVL_MOTION.xCon.SetPosition					:= GVL_MOTION.Script[GVL_MOTION.CurInstruction].SetXPosition - GVL_MOTION.CARRIAGE_OFFSETS[0];
					GVL_MOTION.xCon.SetVelocity					:= GVL_MOTION.Script[GVL_MOTION.CurInstruction].SetXVelocity;
					GVL_MOTION.yCon.SetPosition					:= GVL_MOTION.Script[GVL_MOTION.CurInstruction].SetYPosition - GVL_MOTION.CARRIAGE_OFFSETS[1];
					GVL_MOTION.yCon.SetVelocity					:= GVL_MOTION.Script[GVL_MOTION.CurInstruction].SetYVelocity;
					GVL_MOTION.zCon.SetPosition					:= GVL_MOTION.Script[GVL_MOTION.CurInstruction].SetZPosition - GVL_MOTION.CARRIAGE_OFFSETS[2];
					GVL_MOTION.zCon.SetVelocity					:= GVL_MOTION.Script[GVL_MOTION.CurInstruction].SetZVelocity;
					
					GVL_MOTION.xCon.Execute_MABS				:= TRUE;
					GVL_MOTION.yCon.Execute_MABS				:= TRUE;
					GVL_MOTION.zCon.Execute_MABS				:= TRUE;
				
					GVL_MOTION.InstructionState 				:= 1;	
					
				//outside of basin error	
				ELSE
					GVL_MOTION.STATUS.Basin_Exceed_Err			:= TRUE;
					GVL_MOTION.CurInstruction 					:= 0;
					GVL_MOTION.EXT_CTR.CMDRUN 					:= FALSE;
				END_IF	
				//hard stop error	
// 				ELSE
// 					GVL_MOTION.STATUS.HS_Err					:= TRUE;
// 					GVL_MOTION.STATUS.Move_Abs_Err				:= TRUE;
// 					GVL_MOTION.CurInstruction 					:= 0;
// 					GVL_MOTION.EXT_CTR.CMDRUN 					:= FALSE;
// 				END_IF	
	
			
		ELSIF GVL_MOTION.Script[GVL_MOTION.CurInstruction].MotionCommand = MotionType.Relative THEN
				
				//check hard stops
// 				IF (GVL_MOTION.STATUS.xPosOut + GVL_MOTION.Script[GVL_MOTION.CurInstruction].SetXPosition < GVL_MOTION.STATUS.HardStopLocations[0])
// 				AND(GVL_MOTION.STATUS.yPosOut + GVL_MOTION.Script[GVL_MOTION.CurInstruction].SetXPosition < GVL_MOTION.STATUS.HardStopLocations[1])	
// 				AND(GVL_MOTION.STATUS.zPosOut + GVL_MOTION.Script[GVL_MOTION.CurInstruction].SetXPosition < GVL_MOTION.STATUS.HardStopLocations[2])
// 				THEN
				//check basin
				IF ((GVL_MOTION.Script[GVL_MOTION.CurInstruction].SetXPosition + GVL_MOTION.STATUS.xPosOut) > GVL_MOTION.ActiveBasin.xMin)
				AND((GVL_MOTION.Script[GVL_MOTION.CurInstruction].SetXPosition + GVL_MOTION.STATUS.xPosOut) < GVL_MOTION.ActiveBasin.xMax)	
				AND((GVL_MOTION.Script[GVL_MOTION.CurInstruction].SetYPosition + GVL_MOTION.STATUS.yPosOut) > GVL_MOTION.ActiveBasin.yMin)
				AND((GVL_MOTION.Script[GVL_MOTION.CurInstruction].SetYPosition + GVL_MOTION.STATUS.yPosOut) < GVL_MOTION.ActiveBasin.yMax)
				AND((GVL_MOTION.Script[GVL_MOTION.CurInstruction].SetZPosition + GVL_MOTION.STATUS.zPosOut) > 0)
				AND((GVL_MOTION.Script[GVL_MOTION.CurInstruction].SetZPosition + GVL_MOTION.STATUS.zPosOut) < GVL_MOTION.STATUS.HardStopLocations[2])
				THEN	

					GVL_MOTION.xCon.SetPosition					:= GVL_MOTION.Script[GVL_MOTION.CurInstruction].SetXPosition;
					GVL_MOTION.xCon.SetVelocity					:= GVL_MOTION.Script[GVL_MOTION.CurInstruction].SetXVelocity;
					GVL_MOTION.yCon.SetPosition					:= GVL_MOTION.Script[GVL_MOTION.CurInstruction].SetYPosition;
					GVL_MOTION.yCon.SetVelocity					:= GVL_MOTION.Script[GVL_MOTION.CurInstruction].SetYVelocity;
					GVL_MOTION.zCon.SetPosition					:= GVL_MOTION.Script[GVL_MOTION.CurInstruction].SetZPosition;
					GVL_MOTION.zCon.SetVelocity					:= GVL_MOTION.Script[GVL_MOTION.CurInstruction].SetZVelocity;
				
					
					GVL_MOTION.InstructionState 				:= 1;	
					
				//outside of basin error	
				ELSE
					GVL_MOTION.STATUS.Basin_Exceed_Err			:= TRUE;
					GVL_MOTION.CurInstruction 					:= 0;
					GVL_MOTION.EXT_CTR.CMDRUN 					:= FALSE;
				END_IF	
				//hard stop error	
// 				ELSE
// 					GVL_MOTION.STATUS.HS_Err					:= TRUE;
// 					GVL_MOTION.STATUS.Move_Rel_Err				:= TRUE;
// 					GVL_MOTION.CurInstruction 					:= 0;
// 					GVL_MOTION.EXT_CTR.CMDRUN 					:= FALSE;
// 				END_IF	
			
			
		END_IF	
	
	ELSIF GVL_MOTION.Script[GVL_MOTION.CurInstruction].MotionCommand = MotionType.Time_Wait THEN
		t2(IN := TRUE, PT := GVL_MOTION.Script[GVL_MOTION.CurInstruction].PauseTime);
		GVL_MOTION.InstructionState 							:= 3;
		
	ELSE  
		GVL_MOTION.CurInstruction 								:= 0;
		GVL_MOTION.EXT_CTR.CMDRUN 								:= FALSE; //no queued command means exit
	END_IF

	1:
	//state 1: non DAQ motion
	//button debounce needed coming from pause state 2 or 3
	t5(IN := TRUE, PT := T#30MS);
	IF t5.Q THEN
		
